METHOD PROTECTED FINAL allocate : BOOL
VAR_INPUT
	SizeOfStruct											: 	UDINT;	
END_VAR
IF SizeOfStruct = 0
THEN
	allocate												:= FALSE;
ELSIF pElement_Tmp = 0 
THEN
	pElement_Tmp											:= __NEW(BYTE, SizeOfStruct);
	MemSizeOfStruct											:= SizeOfStruct;
	IF TRUE
	THEN
		AdsLogHint('EngineeringToolbox | FB Quicksort | An instance allocated %s bytes from the dynamic memory of the ADS router memory pool', TO_STRING(MemSizeOfStruct));
	END_IF
	Allocate												:= TRUE;
ELSIF SizeOfStruct > MemSizeOfStruct
THEN
	__DELETE(pElement_Tmp);	
	pElement_Tmp											:= __NEW(BYTE, SizeOfStruct);
	MemSizeOfStruct											:= SizeOfStruct;
		IF TRUE
	THEN
		AdsLogWarn('EngineeringToolbox | FB Quicksort | SizeOfStruct increased and an instance has an additional %s bytes allocated from the dynamic memory of the ADS router memory pool', TO_STRING(MemSizeOfStruct));
	END_IF
	Allocate												:= TRUE;
ELSE
	Allocate												:= TRUE;	
END_IF
END_METHOD

METHOD byDINT : BOOL // returns true if sort ends successfully 
VAR_INPUT
	pData													: 	POINTER TO BYTE := 0;	// ADR(Array) 	
	SizeOfData												: 	UDINT := 0;				// SIZEOF(Array)
	pCompareElement											: 	POINTER TO BYTE := 0;	// ADR(Array[1].DINT)		
	SizeOfStruct											: 	UDINT := 0;				// SIZEOF(Array[1]) 	
END_VAR                                                 
VAR        
	pPivotElement											: 	POINTER TO DINT;		// Pivot value
	PivotElement											: 	DINT;					// Pivot value as DINT	
	pCmpElement												:	POINTER TO DINT;		// compare value
	                                					                            	
	endMainLoop												:	BOOL;					// End of main loop reached
	endSubLoop												:	BOOL;					// End of sub loop reached                                              
	ElementCount											:	DINT;					// No of array elements
	stackCount,left,right,i,j								:	DINT;					// running variables 	
	stack													:	ARRAY[1..32] OF UDINT;	// stack size 32 => ~1 Mio elements *)	
	                                					
	pElement_1												:	POINTER TO BYTE;		// Copy Pointer 1		
	pElement_2												:	POINTER TO BYTE;		// Copy Pointer 2

END_VAR
// ends with true in case of no error	                                    					 					
IF SizeOfStruct = 0 OR SizeOfData = 0
	OR pData = 0 OR pCompareElement = 0
THEN               					                                   					
	byDINT													:= FALSE;
	RETURN;   
ELSE
	byDINT													:= TRUE;                          					
END_IF                                  					
          
// calculate no. of Elements                                
ElementCount												:= TO_DINT(SizeOfData / SizeOfStruct);   		
			
// Quicksort                            					
// initial value of array size          					
left 														:= 1;				// first element
right 														:= ElementCount;	// last element 
stackCount 													:= 1;				// running variable 
                                        	
WHILE NOT endMainLoop DO							
	IF left < right THEN                	
		pPivotElement										:= pCompareElement + (SizeOfStruct * TO_UDINT(SHR(right+left,1)));
		PivotElement										:= pPivotElement^;
		i 													:= left -1;
		j 													:= right +1;
		endSubLoop 											:= FALSE;
		REPEAT
			IF SortInverse
			THEN	// sort descending	
				REPEAT	
					i 										:= i+1;	
					pCmpElement								:= pCompareElement + (SizeOfStruct * TO_UDINT(i-1));
				UNTIL (pCmpElement^ <= PivotElement) OR NOT (i < right)	END_REPEAT	
				REPEAT	
					j 										:= j-1;	
					pCmpElement								:= pCompareElement + (SizeOfStruct * TO_UDINT(j-1));
				UNTIL (pCmpElement^ >= PivotElement) OR NOT (j > left)	END_REPEAT		
			ELSE	// sort ascending
				REPEAT	
					i 										:= i+1;
					pCmpElement								:= pCompareElement + (SizeOfStruct * TO_UDINT(i-1));
				UNTIL (pCmpElement^ >= PivotElement)	OR NOT (i < right)	END_REPEAT;				
				REPEAT	
					j 										:= j-1;	
					pCmpElement								:= pCompareElement + (SizeOfStruct * TO_UDINT(j-1));
				UNTIL (pCmpElement^ <= PivotElement) OR NOT (j > left)	END_REPEAT;
			END_IF
			IF i >= j THEN
				endSubLoop									:= TRUE;
			ELSE                    					
				Allocate( SizeOfStruct);
				pElement_1									:= pData + (SizeOfStruct * TO_UDINT(j-1));
				pElement_2									:= pData + (SizeOfStruct * TO_UDINT(i-1));
				
				IF pElement_Tmp = 0 
					OR_ELSE MEMCPY(pElement_Tmp, pElement_1,	SizeOfStruct) = 0
					OR_ELSE MEMCPY(pElement_1,	pElement_2,		SizeOfStruct) = 0
					OR_ELSE MEMCPY(pElement_2,	pElement_Tmp,	SizeOfStruct) = 0
				THEN
					byDINT									:= FALSE;
					RETURN;	
				END_IF
	
			END_IF
		UNTIL endSubLoop END_REPEAT;		
		stack[stackCount] 									:= TO_UDINT(right); 	// save right in stack			
		IF stackCount < 32              					
		THEN                            					
			stackCount 										:= stackCount +1;
		ELSE															// Error stack Limit    
			endMainLoop 									:= TRUE;
			byDINT											:= FALSE;			
		END_IF                          					
		right 												:= MAX(left, i-1);
	ELSE                                
		IF stackCount = 1 THEN          
			endMainLoop 									:= TRUE;
		ELSE                            					
			left 											:= right+1;       
			stackCount 										:= stackCount -1;	// load from stack
			right											:= TO_DINT(stack[stackCount]);
		END_IF
	END_IF
END_WHILE
END_METHOD

METHOD byDINT_Bubble : BOOL // returns true if sort ends successfully 
VAR_INPUT	
	pData													:	POINTER TO BYTE;// ADR(Array) 			
	SizeOfData												:	UDINT;			// SIZEOF(Array)
	pCompareElement											:	POINTER TO BYTE;// ADR(Array[1].DINT)		
	SizeOfStruct											:	UDINT;			// SIZEOF(Array[1]) 			
END_VAR                                 					                
VAR                                     					                
	Run  													:	DINT;			// main loop
  	Index													:	DINT;			// sub loop 	
	ElementCount											:	DINT;			
	                                    					
	CompareElement_1										:	DINT;					
	CompareElement_2										:	DINT;					
	pCompareElement_1										:	POINTER TO DINT;		
	pCompareElement_2										:	POINTER TO DINT;
		                                					                        
	pElement_1												:	POINTER TO BYTE;		
	pElement_2												:	POINTER TO BYTE;		
END_VAR
// ends with true in case of no error	                                    					 					
IF SizeOfStruct = 0 OR SizeOfData = 0
	OR pData = 0 OR pCompareElement = 0
THEN               					                                   					
	byDINT_Bubble											:= FALSE;
	RETURN;   
ELSE
	byDINT_Bubble											:= TRUE;                          					
END_IF    

// Bubblesort Routine
// Code saving 
	
// calculate no. of Elements                                
ElementCount												:= TO_DINT(SizeOfData / SizeOfStruct);  

// bubblesort 
FOR Run := 1 TO TO_DINT(ElementCount) - 1 DO
    FOR Index := ElementCount - 1 TO Run BY -1 DO
		// get element x for compare 
		pCompareElement_1				:=	pCompareElement + (SizeOfStruct * TO_UDINT(Index));
		CompareElement_1				:=	pCompareElement_1^;
		// get element x-1 for compare 
		pCompareElement_2				:=	pCompareElement + (SizeOfStruct * TO_UDINT(Index-1));
		CompareElement_2 				:=	pCompareElement_2^;
		// switch by useing temporary memory 
		IF ((	CompareElement_1 < CompareElement_2) AND NOT SortInverse)
			OR((CompareElement_1 > CompareElement_2) AND SortInverse)
		THEN
			// get pointer for MEMCPY 
			Allocate(SizeOfStruct);
			pElement_1					:= pData + SizeOfStruct * TO_UDINT(Index);
			pElement_2					:= pData + SizeOfStruct * TO_UDINT(Index-1);
			
	
			IF pElement_Tmp = 0 
				OR_ELSE MEMCPY(pElement_Tmp, pElement_1,	SizeOfStruct) = 0
				OR_ELSE MEMCPY(pElement_1,	pElement_2,		SizeOfStruct) = 0
				OR_ELSE MEMCPY(pElement_2,	pElement_Tmp,	SizeOfStruct) = 0
			THEN
				byDINT_Bubble		:= FALSE;
				EXIT;												
			END_IF

      END_IF
	END_FOR
END_FOR
END_METHOD

METHOD byINT : BOOL // returns true if sort ends successfully 
VAR_INPUT
	pData													: 	POINTER TO BYTE := 0;	// ADR(Array) 	
	SizeOfData												: 	UDINT := 0;				// SIZEOF(Array)
	pCompareElement											: 	POINTER TO BYTE := 0;	// ADR(Array[1].INT)		
	SizeOfStruct											: 	UDINT := 0;				// SIZEOF(Array[1]) 	
END_VAR                                                 
VAR        
	pPivotElement											: 	POINTER TO INT;			// Pivot value
	PivotElement											: 	INT;					// Pivot value as INT	
	pCmpElement												:	POINTER TO INT;			// compare value
	                                					                            	
	endMainLoop												:	BOOL;					// End of main loop reached
	endSubLoop												:	BOOL;					// End of sub loop reached                                              
	ElementCount											:	DINT;					// No of array elements
	stackCount,left,right,i,j								:	DINT;					// running variables 	
	stack													:	ARRAY[1..32] OF UDINT;	// stack size 32 => ~1 Mio elements *)	
	                                					
	pElement_1												:	POINTER TO BYTE;		// Copy Pointer 1		
	pElement_2												:	POINTER TO BYTE;		// Copy Pointer 2
END_VAR
// ends with true in case of no error	                                    					 					
IF SizeOfStruct = 0 OR SizeOfData = 0
	OR pData = 0 OR pCompareElement = 0
THEN               					                                   					
	byINT													:= FALSE;
	RETURN;   
ELSE
	byINT													:= TRUE;                          					
END_IF                                    					
        
// calculate no. of Elements                                
ElementCount												:= TO_DINT(SizeOfData / SizeOfStruct);   
                                					
// Quicksort                            					
// initial value of array size          					
left 														:= 1;				// first element
right 														:= ElementCount;	// last element 
stackCount 													:= 1;				// running variable 
                                        	
WHILE NOT endMainLoop DO							
	IF left < right THEN                	
		pPivotElement										:= pCompareElement + (SizeOfStruct * TO_UDINT(SHR(right+left,1)));
		PivotElement										:= pPivotElement^;
		i 													:= left -1;
		j 													:= right +1;
		endSubLoop 											:= FALSE;
		REPEAT
			IF SortInverse
			THEN	// sort descending	
				REPEAT	
					i 										:= i+1;	
					pCmpElement								:= pCompareElement + (SizeOfStruct * TO_UDINT(i-1));
				UNTIL (pCmpElement^ <= PivotElement) OR NOT (i < right)	END_REPEAT	
				REPEAT	
					j 										:= j-1;	
					pCmpElement								:= pCompareElement + (SizeOfStruct * TO_UDINT(j-1));
				UNTIL (pCmpElement^ >= PivotElement) OR NOT (j > left)	END_REPEAT		
			ELSE	// sort ascending
				REPEAT	
					i 										:= i+1;
					pCmpElement								:= pCompareElement + (SizeOfStruct * TO_UDINT(i-1));
				UNTIL (pCmpElement^ >= PivotElement)	OR NOT (i < right)	END_REPEAT;				
				REPEAT	
					j 										:= j-1;	
					pCmpElement								:= pCompareElement + (SizeOfStruct * TO_UDINT(j-1));
				UNTIL (pCmpElement^ <= PivotElement) OR NOT (j > left)	END_REPEAT;
			END_IF
			IF i >= j THEN
				endSubLoop									:= TRUE;
			ELSE                    					
				Allocate(SizeOfStruct);
				pElement_1									:= pData + (SizeOfStruct * TO_UDINT(j-1));
				pElement_2									:= pData + (SizeOfStruct * TO_UDINT(i-1));
				
				IF pElement_Tmp = 0 
					OR_ELSE MEMCPY(pElement_Tmp, pElement_1,	SizeOfStruct) = 0
					OR_ELSE MEMCPY(pElement_1,	pElement_2,		SizeOfStruct) = 0
					OR_ELSE MEMCPY(pElement_2,	pElement_Tmp,	SizeOfStruct) = 0
				THEN
					byINT									:= FALSE;
					RETURN;	
				END_IF
	
			END_IF
		UNTIL endSubLoop END_REPEAT;		
		stack[stackCount] 									:= TO_UDINT(right); 	// save right in stack			
		IF stackCount < 32              					
		THEN                            					
			stackCount 										:= stackCount +1;
		ELSE															// Error stack Limit    
			endMainLoop 									:= TRUE;
			byINT											:= FALSE;			
		END_IF                          					
		right 												:= MAX(left, i-1);
	ELSE                                
		IF stackCount = 1 THEN          
			endMainLoop 									:= TRUE;
		ELSE                            					
			left 											:= right+1;       
			stackCount 										:= stackCount -1;	// load from stack
			right											:= TO_DINT(stack[stackCount]);
		END_IF
	END_IF
END_WHILE
END_METHOD

METHOD byLREAL : BOOL // returns true if sort ends successfully 
VAR_INPUT
	pData													: 	POINTER TO BYTE := 0;	// ADR(Array) 	
	SizeOfData												: 	UDINT := 0;				// SIZEOF(Array)
	pCompareElement											: 	POINTER TO BYTE := 0;	// ADR(Array[1].LREAL)		
	SizeOfStruct											: 	UDINT := 0;				// SIZEOF(Array[1]) 	
END_VAR                                                 
VAR        
	pPivotElement											: 	POINTER TO LREAL;		// Pivot value	
	PivotElement											: 	LREAL;					// Pivot value as LREAL
	pCmpElement												:	POINTER TO LREAL;		// compare value
	                                					                            	
	endMainLoop												:	BOOL;					// End of main loop reached
	endSubLoop												:	BOOL;					// End of sub loop reached                                              
	ElementCount											:	DINT;					// No of array elements
	stackCount,left,right,i,j								:	DINT;					// running variables 	
	stack													:	ARRAY[1..32] OF UDINT;	// stack size 32 => ~1 Mio elements *)	
	                                					
	pElement_1												:	POINTER TO BYTE;		// Copy Pointer 1		
	pElement_2												:	POINTER TO BYTE;		// Copy Pointer 2
	
END_VAR
// ends with true in case of no error	                                    					 					
IF SizeOfStruct = 0 OR SizeOfData = 0
	OR pData = 0 OR pCompareElement = 0
THEN               					                                   					
	byLREAL													:= FALSE;
	RETURN;   
ELSE
	byLREAL													:= TRUE;                          					
END_IF                                 					
            
// calculate no. of Elements                                
ElementCount												:= TO_DINT(SizeOfData / SizeOfStruct);   
                            					
// Quicksort                            					
// initial value of array size          					
left 														:= 1;				// first element
right 														:= ElementCount;	// last element 
stackCount 													:= 1;				// running variable 
                                        	
WHILE NOT endMainLoop DO							
	IF left < right THEN                	
		pPivotElement										:= pCompareElement + (SizeOfStruct * TO_UDINT(SHR(right+left,1))); // divide by 2
		PivotElement										:= pPivotElement^;
		i 													:= left -1;
		j 													:= right +1;
		endSubLoop 											:= FALSE;
		REPEAT
			IF SortInverse
			THEN	// sort descending	
				REPEAT	
					i 										:= i+1;	
					pCmpElement								:= pCompareElement + (SizeOfStruct * TO_UDINT(i-1));
				UNTIL (pCmpElement^ <= PivotElement) OR NOT (i < right)	END_REPEAT	
				REPEAT	
					j 										:= j-1;	
					pCmpElement								:= pCompareElement + (SizeOfStruct * TO_UDINT(j-1));
				UNTIL (pCmpElement^ >= PivotElement) OR NOT (j > left)	END_REPEAT		
			ELSE	// sort ascending
				REPEAT	
					i 										:= i+1;
					pCmpElement								:= pCompareElement + (SizeOfStruct * TO_UDINT(i-1));
				UNTIL (pCmpElement^ >= PivotElement)	OR NOT (i < right)	END_REPEAT;				
				REPEAT	
					j 										:= j-1;	
					pCmpElement								:= pCompareElement + (SizeOfStruct * TO_UDINT(j-1));
				UNTIL (pCmpElement^ <= PivotElement) OR NOT (j > left)	END_REPEAT;
			END_IF
			IF i >= j THEN
				endSubLoop									:= TRUE;
			ELSE                    					
				Allocate(SizeOfStruct);
				pElement_1									:= pData + (SizeOfStruct * TO_UDINT(j-1));
				pElement_2									:= pData + (SizeOfStruct * TO_UDINT(i-1));
				
				IF pElement_Tmp = 0 
					OR_ELSE MEMCPY(pElement_Tmp, pElement_1,	SizeOfStruct) = 0
					OR_ELSE MEMCPY(pElement_1,	pElement_2,		SizeOfStruct) = 0
					OR_ELSE MEMCPY(pElement_2,	pElement_Tmp,	SizeOfStruct) = 0
				THEN
					byLREAL									:= FALSE;
					RETURN;	
				END_IF

			END_IF
		UNTIL endSubLoop END_REPEAT;		
		stack[stackCount] 									:= TO_UDINT(right); 	// save right in stack			
		IF stackCount < 32              					
		THEN                            					
			stackCount 										:= stackCount +1;
		ELSE															// Error stack Limit    
			endMainLoop 									:= TRUE;
			byLREAL											:= FALSE;			
		END_IF                          					
		right 												:= MAX(left, i-1);
	ELSE                                
		IF stackCount = 1 THEN          
			endMainLoop 									:= TRUE;
		ELSE                            					
			left 											:= right+1;       
			stackCount 										:= stackCount -1;	// load from stack
			right											:= TO_DINT(stack[stackCount]);
		END_IF
	END_IF
END_WHILE
END_METHOD

METHOD byLTIME : BOOL // returns true if sort ends successfully 
VAR_INPUT
	pData													: 	POINTER TO BYTE := 0;	// ADR(Array) 	
	SizeOfData												: 	UDINT := 0;				// SIZEOF(Array)
	pCompareElement											: 	POINTER TO BYTE := 0;	// ADR(Array[1].LTIME)		
	SizeOfStruct											: 	UDINT := 0;				// SIZEOF(Array[1]) 	
END_VAR                                                 
VAR        
	pPivotElement											: 	POINTER TO LTIME;		// Pivot value	
	PivotElement											: 	LTIME;					// Pivot value as LTIME	
	pCmpElement												:	POINTER TO LTIME;		// compare value
	                                					                            	
	endMainLoop												:	BOOL;					// End of main loop reached
	endSubLoop												:	BOOL;					// End of sub loop reached                                              
	ElementCount											:	DINT;					// No of array elements
	stackCount,left,right,i,j								:	DINT;					// running variables 	
	stack													:	ARRAY[1..32] OF UDINT;	// stack size 32 => ~1 Mio elements *)	
	                                					
	pElement_1												:	POINTER TO BYTE;		// Copy Pointer 1		
	pElement_2												:	POINTER TO BYTE;		// Copy Pointer 2
END_VAR
// ends with true in case of no error	                                    					 					
IF SizeOfStruct = 0 OR SizeOfData = 0
	OR pData = 0 OR pCompareElement = 0
THEN               					                                   					
	byLTIME													:= FALSE;
	RETURN;   
ELSE
	byLTIME													:= TRUE;                          					
END_IF                                    					
             
// calculate no. of Elements                                
ElementCount												:= TO_DINT(SizeOfData / SizeOfStruct);   
                           					
// Quicksort                            					
// initial value of array size          					
left 														:= 1;				// first element
right 														:= ElementCount;	// last element 
stackCount 													:= 1;				// running variable 
                                        	
WHILE NOT endMainLoop DO							
	IF left < right THEN                	
		pPivotElement										:= pCompareElement + (SizeOfStruct * TO_UDINT(SHR(right+left,1)));
		PivotElement										:= pPivotElement^;
		i 													:= left -1;
		j 													:= right +1;
		endSubLoop 											:= FALSE;
		REPEAT
			IF SortInverse
			THEN	// sort descending	
				REPEAT	
					i 										:= i+1;	
					pCmpElement								:= pCompareElement + (SizeOfStruct * TO_UDINT(i-1));
				UNTIL (pCmpElement^ <= PivotElement) OR NOT (i < right)	END_REPEAT	
				REPEAT	
					j 										:= j-1;	
					pCmpElement								:= pCompareElement + (SizeOfStruct * TO_UDINT(j-1));
				UNTIL (pCmpElement^ >= PivotElement) OR NOT (j > left)	END_REPEAT		
			ELSE	// sort ascending
				REPEAT	
					i 										:= i+1;
					pCmpElement								:= pCompareElement + (SizeOfStruct * TO_UDINT(i-1));
				UNTIL (pCmpElement^ >= PivotElement)	OR NOT (i < right)	END_REPEAT;				
				REPEAT	
					j 										:= j-1;	
					pCmpElement								:= pCompareElement + (SizeOfStruct * TO_UDINT(j-1));
				UNTIL (pCmpElement^ <= PivotElement) OR NOT (j > left)	END_REPEAT;
			END_IF
			IF i >= j THEN
				endSubLoop									:= TRUE;
			ELSE                    					
				Allocate(SizeOfStruct);
				pElement_1									:= pData + (SizeOfStruct * TO_UDINT(j-1));
				pElement_2									:= pData + (SizeOfStruct * TO_UDINT(i-1));
				
				IF pElement_Tmp = 0 
					OR_ELSE MEMCPY(pElement_Tmp, pElement_1,	SizeOfStruct) = 0
					OR_ELSE MEMCPY(pElement_1,	pElement_2,		SizeOfStruct) = 0
					OR_ELSE MEMCPY(pElement_2,	pElement_Tmp,	SizeOfStruct) = 0
				THEN
					byLTIME									:= FALSE;
					RETURN;	
				END_IF

			END_IF
		UNTIL endSubLoop END_REPEAT;		
		stack[stackCount] 									:= TO_UDINT(right); 	// save right in stack			
		IF stackCount < 32              					
		THEN                            					
			stackCount 										:= stackCount +1;
		ELSE															// Error stack Limit    
			endMainLoop 									:= TRUE;
			byLTIME											:= FALSE;			
		END_IF                          					
		right 												:= MAX(left, i-1);
	ELSE                                
		IF stackCount = 1 THEN          
			endMainLoop 									:= TRUE;
		ELSE                            					
			left 											:= right+1;       
			stackCount 										:= stackCount -1;	// load from stack
			right											:= TO_DINT(stack[stackCount]);
		END_IF
	END_IF
END_WHILE
END_METHOD

METHOD byREAL : BOOL // returns true if sort ends successfully 
VAR_INPUT
	pData													: 	POINTER TO BYTE := 0;	// ADR(Array) 	
	SizeOfData												: 	UDINT := 0;				// SIZEOF(Array)
	pCompareElement											: 	POINTER TO BYTE := 0;	// ADR(Array[1].REAL)		
	SizeOfStruct											: 	UDINT := 0;				// SIZEOF(Array[1]) 	
END_VAR                                                 
VAR        
	pPivotElement											: 	POINTER TO REAL;		// Pivot value	
	PivotElement											: 	REAL;					// Pivot value as REAL	
	pCmpElement												:	POINTER TO REAL;		// compare value
	                                					                            	
	endMainLoop												:	BOOL;					// End of main loop reached
	endSubLoop												:	BOOL;					// End of sub loop reached                                              
	ElementCount											:	DINT;					// No of array elements
	stackCount,left,right,i,j								:	DINT;					// running variables 	
	stack													:	ARRAY[1..32] OF UDINT;	// stack size 32 => ~1 Mio elements *)	
	                                					
	pElement_1												:	POINTER TO BYTE;		// Copy Pointer 1		
	pElement_2												:	POINTER TO BYTE;		// Copy Pointer 2
END_VAR
// ends with true in case of no error	                                    					 					
IF SizeOfStruct = 0 OR SizeOfData = 0
	OR pData = 0 OR pCompareElement = 0
THEN               					                                   					
	byREAL													:= FALSE;
	RETURN;   
ELSE
	byREAL													:= TRUE;                          					
END_IF                                   					
          
// calculate no. of Elements                                
ElementCount												:= TO_DINT(SizeOfData / SizeOfStruct);   
                              					
// Quicksort                            					
// initial value of array size          					
left 														:= 1;				// first element
right 														:= ElementCount;	// last element 
stackCount 													:= 1;				// running variable 
                                        	
WHILE NOT endMainLoop DO							
	IF left < right THEN                	
		pPivotElement										:= pCompareElement + (SizeOfStruct * TO_UDINT(SHR(right+left,1)));
		PivotElement										:= pPivotElement^;
		i 													:= left -1;
		j 													:= right +1;
		endSubLoop 											:= FALSE;
		REPEAT
			IF SortInverse
			THEN	// sort descending	
				REPEAT	
					i 										:= i+1;	
					pCmpElement								:= pCompareElement + (SizeOfStruct * TO_UDINT(i-1));
				UNTIL (pCmpElement^ <= PivotElement) OR NOT (i < right)	END_REPEAT	
				REPEAT	
					j 										:= j-1;	
					pCmpElement								:= pCompareElement + (SizeOfStruct * TO_UDINT(j-1));
				UNTIL (pCmpElement^ >= PivotElement) OR NOT (j > left)	END_REPEAT		
			ELSE	// sort ascending
				REPEAT	
					i 										:= i+1;
					pCmpElement								:= pCompareElement + (SizeOfStruct * TO_UDINT(i-1));
				UNTIL (pCmpElement^ >= PivotElement)	OR NOT (i < right)	END_REPEAT;				
				REPEAT	
					j 										:= j-1;	
					pCmpElement								:= pCompareElement + (SizeOfStruct * TO_UDINT(j-1));
				UNTIL (pCmpElement^ <= PivotElement) OR NOT (j > left)	END_REPEAT;
			END_IF
			IF i >= j THEN
				endSubLoop									:= TRUE;
			ELSE                    					
				Allocate(SizeOfStruct);
				pElement_1									:= pData + (SizeOfStruct * TO_UDINT(j-1));
				pElement_2									:= pData + (SizeOfStruct * TO_UDINT(i-1));
				
				IF pElement_Tmp = 0 
					OR_ELSE MEMCPY(pElement_Tmp, pElement_1,	SizeOfStruct) = 0
					OR_ELSE MEMCPY(pElement_1,	pElement_2,		SizeOfStruct) = 0
					OR_ELSE MEMCPY(pElement_2,	pElement_Tmp,	SizeOfStruct) = 0
				THEN
					byREAL									:= FALSE;
					RETURN;	
				END_IF

			END_IF
		UNTIL endSubLoop END_REPEAT;		
		stack[stackCount] 									:= TO_UDINT(right); 	// save right in stack			
		IF stackCount < 32              					
		THEN                            					
			stackCount 										:= stackCount +1;
		ELSE															// Error stack Limit    
			endMainLoop 									:= TRUE;
			byREAL											:= FALSE;			
		END_IF                          					
		right 												:= MAX(left, i-1);
	ELSE                                
		IF stackCount = 1 THEN          
			endMainLoop 									:= TRUE;
		ELSE                            					
			left 											:= right+1;       
			stackCount 										:= stackCount -1;	// load from stack
			right											:= TO_DINT(stack[stackCount]);
		END_IF
	END_IF
END_WHILE
END_METHOD

METHOD bySTRING : BOOL // returns true if sort ends successfully 
VAR_INPUT
	pData													: 	POINTER TO BYTE := 0;	// ADR(Array) 	
	SizeOfData												: 	UDINT := 0;				// SIZEOF(Array)
	pCompareElement											: 	POINTER TO BYTE := 0;	// ADR(Array[1].STRING)		
	SizeOfStruct											: 	UDINT := 0;				// SIZEOF(Array[1]) 	
END_VAR                                                                                        
VAR        
	pPivotElement											: 	POINTER TO STRING(MAX_STRING_LENGTH);	// Pivot value
	pCmpElement												:	POINTER TO STRING(MAX_STRING_LENGTH);	// compare value
	PivotElement											:	BYTE; 					// Pivot value	
	CompareElement											:	BYTE; 					// compare value
                               					                            	
	endMainLoop												:	BOOL;					// End of main loop reached
	endSubLoop												:	BOOL;					// End of sub loop reached                                              
	ElementCount											:	DINT;					// No of array elements
	stackCount,left,right,i,j,k								:	DINT;					// running variables 	
	stack													:	ARRAY[1..32] OF UDINT;	// stack size 32 => ~1 Mio elements *)	
	                                					
	pElement_1												:	POINTER TO BYTE;		// Copy Pointer 1		
	pElement_2												:	POINTER TO BYTE;		// Copy Pointer 2
END_VAR
// ends with true in case of no error	                                    					 					
IF SizeOfStruct = 0 OR SizeOfData = 0
	OR pData = 0 OR pCompareElement = 0
THEN               					                                   					
	bySTRING												:= FALSE;
	RETURN;   
ELSE
	bySTRING												:= TRUE;                          					
END_IF                                 					
          
// calculate no. of Elements                                
ElementCount												:= TO_DINT(SizeOfData / SizeOfStruct);   
                              					
// Quicksort                            					
// initial value of array size          					
left 														:= 1;				// first element
right 														:= ElementCount;	// last element 
stackCount 													:= 1;				// running variable 
                                        	
WHILE NOT endMainLoop DO							
	IF left < right THEN                	
		pPivotElement										:= pCompareElement + (SizeOfStruct * TO_UDINT(SHR(right+left,1)));
		i 													:= left -1;
		j 													:= right +1;
		endSubLoop 											:= FALSE;
		REPEAT
			IF SortInverse
			THEN	// sort descending	
				REPEAT	
					i 										:= i+1;	
					pCmpElement								:= pCompareElement + (SizeOfStruct * TO_UDINT(i-1));
					FOR k := 1 TO MAX_STRING_LENGTH DO // Find unequal char
						// element 1,2 to upper char 	https://www.uni-due.de/hummell/infos/ascii/
						IF pCmpElement^[k] = 0 
							AND IgnoreBlank
						THEN
							CompareElement					:= 127;
						ELSE
							CompareElement					:= SEL(pCmpElement^[k] >= 97(*a*)	AND_THEN pCmpElement^[k] <= 122(*z*), 	pCmpElement^[k],pCmpElement^[k] - 32);		// a --> A
						END_IF						
						IF pPivotElement^[k] = 0 
							AND IgnoreBlank
						THEN
							PivotElement					:= 127;
						ELSE
							PivotElement					:= SEL(pPivotElement^[k] >= 97(*a*) AND_THEN pPivotElement^[k] <= 122(*z*), pPivotElement^[k], 	pPivotElement^[k] - 32);// a --> A
						END_IF
						// Find unequal char
						IF CompareElement <> PivotElement
							OR CompareElement = 0
							OR PivotElement = 0
						THEN
							EXIT;
						END_IF
					END_FOR
				UNTIL (CompareElement <= PivotElement) OR NOT (i < right)	END_REPEAT	
				REPEAT	
					j 										:= j-1;	
					pCmpElement								:= pCompareElement + (SizeOfStruct * TO_UDINT(j-1));
					FOR k := 0 TO MAX_STRING_LENGTH DO // Find unequal char
						// element 1,2 to upper char 	https://www.uni-due.de/hummell/infos/ascii/
						IF pCmpElement^[k] = 0 
							AND IgnoreBlank
						THEN
							CompareElement					:= 127;
						ELSE
							CompareElement					:= SEL(pCmpElement^[k] >= 97(*a*)	AND_THEN pCmpElement^[k] <= 122(*z*), 	pCmpElement^[k],pCmpElement^[k] - 32);		// a --> A
						END_IF
						IF pPivotElement^[k] = 0 
							AND IgnoreBlank
						THEN
							PivotElement					:= 127;
						ELSE
							PivotElement					:= SEL(pPivotElement^[k] >= 97(*a*) AND_THEN pPivotElement^[k] <= 122(*z*), pPivotElement^[k], 	pPivotElement^[k] - 32);// a --> A
						END_IF
						// Find unequal char
						IF CompareElement <> PivotElement
							OR CompareElement = 0
							OR PivotElement = 0
						THEN
							EXIT;
						END_IF
					END_FOR
				UNTIL (CompareElement >= PivotElement) OR NOT (j > left)	END_REPEAT		
			ELSE	// sort ascending
				REPEAT	
					i 										:= i+1;
					pCmpElement								:= pCompareElement + (SizeOfStruct * TO_UDINT(i-1));
					FOR k := 0 TO MAX_STRING_LENGTH DO // Find unequal char
						// element 1,2 to upper char 	https://www.uni-due.de/hummell/infos/ascii/
						IF pCmpElement^[k] = 0 
							AND IgnoreBlank
						THEN
							CompareElement					:= 127;
						ELSE
							CompareElement					:= SEL(pCmpElement^[k] >= 97(*a*)	AND_THEN pCmpElement^[k] <= 122(*z*), 	pCmpElement^[k],pCmpElement^[k] - 32);		// a --> A
						END_IF
						IF pPivotElement^[k] = 0 
							AND IgnoreBlank
						THEN
							PivotElement					:= 127;
						ELSE
							PivotElement					:= SEL(pPivotElement^[k] >= 97(*a*) AND_THEN pPivotElement^[k] <= 122(*z*), pPivotElement^[k], 	pPivotElement^[k] - 32);// a --> A
						END_IF
						// Find unequal char
						IF CompareElement <> PivotElement
							OR CompareElement = 0
							OR PivotElement = 0
						THEN
							EXIT;
						END_IF
					END_FOR
				UNTIL (CompareElement >= PivotElement)	OR NOT (i < right)	END_REPEAT;				
				REPEAT	
					j 										:= j-1;	
					pCmpElement								:= pCompareElement + (SizeOfStruct * TO_UDINT(j-1));
					FOR k := 0 TO MAX_STRING_LENGTH DO // Find unequal char
						// element 1,2 to upper char 	https://www.uni-due.de/hummell/infos/ascii/
						IF pCmpElement^[k] = 0 
							AND IgnoreBlank
						THEN	
							CompareElement					:= 127;
						ELSE
							CompareElement					:= SEL(pCmpElement^[k] >= 97(*a*)	AND_THEN pCmpElement^[k] <= 122(*z*), 	pCmpElement^[k],pCmpElement^[k] - 32);		// a --> A
						END_IF
						IF pPivotElement^[k] = 0
							AND IgnoreBlank 
						THEN
							PivotElement					:= 127;
						ELSE
							PivotElement					:= SEL(pPivotElement^[k] >= 97(*a*) AND_THEN pPivotElement^[k] <= 122(*z*), pPivotElement^[k], 	pPivotElement^[k] - 32);// a --> A
						END_IF
						// Find unequal char
						IF CompareElement <> PivotElement
							OR CompareElement = 0
							OR PivotElement = 0
						THEN
							EXIT;
						END_IF
					END_FOR
				UNTIL (CompareElement <= PivotElement) OR NOT (j > left)	END_REPEAT;
			END_IF
			IF i >= j THEN
				endSubLoop									:= TRUE;
			ELSE                    					
				Allocate(SizeOfStruct);
				pElement_1									:= pData + (SizeOfStruct * TO_UDINT(j-1));
				pElement_2									:= pData + (SizeOfStruct * TO_UDINT(i-1));
				
				IF pElement_Tmp = 0 
					OR_ELSE MEMCPY(pElement_Tmp, pElement_1,	SizeOfStruct) = 0
					OR_ELSE MEMCPY(pElement_1,	pElement_2,		SizeOfStruct) = 0
					OR_ELSE MEMCPY(pElement_2,	pElement_Tmp,	SizeOfStruct) = 0
				THEN
					bySTRING								:= FALSE;
					RETURN;	
				END_IF

			END_IF
		UNTIL endSubLoop END_REPEAT;		
		stack[stackCount] 									:= TO_UDINT(right); 	// save right in stack			
		IF stackCount < 32              					
		THEN                            					
			stackCount 										:= stackCount +1;
		ELSE															// Error stack Limit    
			endMainLoop 									:= TRUE;
			bySTRING										:= FALSE;			
		END_IF                          					
		right 												:= MAX(left, i-1);
	ELSE                                
		IF stackCount = 1 THEN          
			endMainLoop 									:= TRUE;
		ELSE                            					
			left 											:= right+1;       
			stackCount 										:= stackCount -1;	// load from stack
			right											:= TO_DINT(stack[stackCount]);
		END_IF
	END_IF
END_WHILE
END_METHOD

METHOD byTIME : BOOL // returns true if sort ends successfully 
VAR_INPUT
	pData													: 	POINTER TO BYTE := 0;	// ADR(Array) 	
	SizeOfData												: 	UDINT := 0;				// SIZEOF(Array)
	pCompareElement											: 	POINTER TO BYTE := 0;	// ADR(Array[1].TIME)		
	SizeOfStruct											: 	UDINT := 0;				// SIZEOF(Array[1]) 	
END_VAR                                                 
VAR        
	pPivotElement											: 	POINTER TO TIME;		// Pivot value
	PivotElement											: 	TIME;					// Pivot value as TIME	
	pCmpElement												:	POINTER TO TIME;		// compare value
	                                					                            	
	endMainLoop												:	BOOL;					// End of main loop reached
	endSubLoop												:	BOOL;					// End of sub loop reached                                              
	ElementCount											:	DINT;					// No of array elements
	stackCount,left,right,i,j								:	DINT;					// running variables 	
	stack													:	ARRAY[1..32] OF UDINT;	// stack size 32 => ~1 Mio elements *)	
	                                					
	pElement_1												:	POINTER TO BYTE;		// Copy Pointer 1		
	pElement_2												:	POINTER TO BYTE;		// Copy Pointer 2
END_VAR
// ends with true in case of no error	                                    					 					
IF SizeOfStruct = 0 OR SizeOfData = 0
	OR pData = 0 OR pCompareElement = 0
THEN               					                                   					
	byTIME													:= FALSE;
	RETURN;   
ELSE
	byTIME													:= TRUE;                          					
END_IF   

// calculate no. of Elements                                
ElementCount												:= TO_DINT(SizeOfData / SizeOfStruct);                                   					
                                        					
// Quicksort                            					
// initial value of array size          					
left 														:= 1;				// first element
right 														:= ElementCount;	// last element 
stackCount 													:= 1;				// running variable 
                                        	
WHILE NOT endMainLoop DO							
	IF left < right THEN                	
		pPivotElement										:= pCompareElement + (SizeOfStruct * TO_UDINT(SHR(right+left,1)));
		PivotElement										:= pPivotElement^;
		i 													:= left -1;
		j 													:= right +1;
		endSubLoop 											:= FALSE;
		REPEAT
			IF SortInverse
			THEN	// sort descending	
				REPEAT	
					i 										:= i+1;	
					pCmpElement								:= pCompareElement + (SizeOfStruct * TO_UDINT(i-1));
				UNTIL (pCmpElement^ <= PivotElement) OR NOT (i < right)	END_REPEAT	
				REPEAT	
					j 										:= j-1;	
					pCmpElement								:= pCompareElement + (SizeOfStruct * TO_UDINT(j-1));
				UNTIL (pCmpElement^ >= PivotElement) OR NOT (j > left)	END_REPEAT		
			ELSE	// sort ascending
				REPEAT	
					i 										:= i+1;
					pCmpElement								:= pCompareElement + (SizeOfStruct * TO_UDINT(i-1));
				UNTIL (pCmpElement^ >= PivotElement)	OR NOT (i < right)	END_REPEAT;				
				REPEAT	
					j 										:= j-1;	
					pCmpElement								:= pCompareElement + (SizeOfStruct * TO_UDINT(j-1));
				UNTIL (pCmpElement^ <= PivotElement) OR NOT (j > left)	END_REPEAT;
			END_IF
			IF i >= j THEN
				endSubLoop									:= TRUE;
			ELSE                    					
				Allocate(SizeOfStruct);
				pElement_1									:= pData + (SizeOfStruct * TO_UDINT(j-1));
				pElement_2									:= pData + (SizeOfStruct * TO_UDINT(i-1));
				
				IF pElement_Tmp = 0 
					OR_ELSE MEMCPY(pElement_Tmp, pElement_1,	SizeOfStruct) = 0
					OR_ELSE MEMCPY(pElement_1,	pElement_2,		SizeOfStruct) = 0
					OR_ELSE MEMCPY(pElement_2,	pElement_Tmp,	SizeOfStruct) = 0
				THEN
					byTIME									:= FALSE;
					RETURN;	
				END_IF

			END_IF
		UNTIL endSubLoop END_REPEAT;		
		stack[stackCount] 									:= TO_UDINT(right); 	// save right in stack			
		IF stackCount < 32              					
		THEN                            					
			stackCount 										:= stackCount +1;
		ELSE															// Error stack Limit    
			endMainLoop 									:= TRUE;
			byTIME											:= FALSE;			
		END_IF                          					
		right 												:= MAX(left, i-1);
	ELSE                                
		IF stackCount = 1 THEN          
			endMainLoop 									:= TRUE;
		ELSE                            					
			left 											:= right+1;       
			stackCount 										:= stackCount -1;	// load from stack
			right											:= TO_DINT(stack[stackCount]);
		END_IF
	END_IF
END_WHILE
END_METHOD

METHOD byUINT : BOOL // returns true if sort ends successfully 
VAR_INPUT
	pData													: 	POINTER TO BYTE := 0;	// ADR(Array) 	
	SizeOfData												: 	UDINT := 0;				// SIZEOF(Array)
	pCompareElement											: 	POINTER TO BYTE := 0;	// ADR(Array[1].UINT)		
	SizeOfStruct											: 	UDINT := 0;				// SIZEOF(Array[1]) 	
END_VAR                                                 
VAR        
	pPivotElement											: 	POINTER TO UINT;		// Pivot value	
	PivotElement											: 	UINT;					// Pivot value as UINT	
	pCmpElement												:	POINTER TO UINT;		// compare value
	                                					                            	
	endMainLoop												:	BOOL;					// End of main loop reached
	endSubLoop												:	BOOL;					// End of sub loop reached                                              
	ElementCount											:	DINT;					// No of array elements
	stackCount,left,right,i,j								:	DINT;					// running variables 	
	stack													:	ARRAY[1..32] OF UDINT;	// stack size 32 => ~1 Mio elements *)	
	                                					
	pElement_1												:	POINTER TO BYTE;		// Copy Pointer 1		
	pElement_2												:	POINTER TO BYTE;		// Copy Pointer 2
END_VAR
// ends with true in case of no error	                                    					 					
IF SizeOfStruct = 0 OR SizeOfData = 0
	OR pData = 0 OR pCompareElement = 0
THEN               					                                   					
	byUINT													:= FALSE;
	RETURN;   
ELSE
	byUINT													:= TRUE;                          					
END_IF     

// calculate no. of Elements                                
ElementCount												:= TO_DINT(SizeOfData / SizeOfStruct);                                 					
                                        					
// Quicksort                            					
// initial value of array size          					
left 														:= 1;				// first element
right 														:= ElementCount;	// last element 
stackCount 													:= 1;				// running variable 
                                        	
WHILE NOT endMainLoop DO							
	IF left < right THEN                	
		pPivotElement										:= pCompareElement + (SizeOfStruct * TO_UDINT(SHR(right+left,1)));
		PivotElement										:= pPivotElement^;
		i 													:= left -1;
		j 													:= right +1;
		endSubLoop 											:= FALSE;
		REPEAT
			IF SortInverse
			THEN	// sort descending	
				REPEAT	
					i 										:= i+1;	
					pCmpElement								:= pCompareElement + (SizeOfStruct * TO_UDINT(i-1));
				UNTIL (pCmpElement^ <= PivotElement) OR NOT (i < right)	END_REPEAT	
				REPEAT	
					j 										:= j-1;	
					pCmpElement								:= pCompareElement + (SizeOfStruct * TO_UDINT(j-1));
				UNTIL (pCmpElement^ >= PivotElement) OR NOT (j > left)	END_REPEAT		
			ELSE	// sort ascending
				REPEAT	
					i 										:= i+1;
					pCmpElement								:= pCompareElement + (SizeOfStruct * TO_UDINT(i-1));
				UNTIL (pCmpElement^ >= PivotElement)	OR NOT (i < right)	END_REPEAT;				
				REPEAT	
					j 										:= j-1;	
					pCmpElement								:= pCompareElement + (SizeOfStruct * TO_UDINT(j-1));
				UNTIL (pCmpElement^ <= PivotElement) OR NOT (j > left)	END_REPEAT;
			END_IF
			IF i >= j THEN
				endSubLoop									:= TRUE;
			ELSE                    					
				Allocate(SizeOfStruct);
				pElement_1									:= pData + (SizeOfStruct * TO_UDINT(j-1));
				pElement_2									:= pData + (SizeOfStruct * TO_UDINT(i-1));
				
				IF pElement_Tmp = 0 
					OR_ELSE MEMCPY(pElement_Tmp, pElement_1,	SizeOfStruct) = 0
					OR_ELSE MEMCPY(pElement_1,	pElement_2,		SizeOfStruct) = 0
					OR_ELSE MEMCPY(pElement_2,	pElement_Tmp,	SizeOfStruct) = 0
				THEN
					byUINT									:= FALSE;
					RETURN;	
				END_IF

			END_IF
		UNTIL endSubLoop END_REPEAT;		
		stack[stackCount] 									:= TO_UDINT(right); 	// save right in stack			
		IF stackCount < 32              					
		THEN                            					
			stackCount 										:= stackCount +1;
		ELSE															// Error stack Limit    
			endMainLoop 									:= TRUE;
			byUINT											:= FALSE;			
		END_IF                          					
		right 												:= MAX(left, i-1);
	ELSE                                
		IF stackCount = 1 THEN          
			endMainLoop 									:= TRUE;
		ELSE                            					
			left 											:= right+1;       
			stackCount 										:= stackCount -1;	// load from stack
			right											:= TO_DINT(stack[stackCount]);
		END_IF
	END_IF
END_WHILE
END_METHOD

METHOD byUSINT : BOOL // returns true if sort ends successfully 
VAR_INPUT
	pData													: 	POINTER TO BYTE := 0;	// ADR(Array) 	
	SizeOfData												: 	UDINT := 0;				// SIZEOF(Array)
	pCompareElement											: 	POINTER TO BYTE := 0;	// ADR(Array[1].USINT)		
	SizeOfStruct											: 	UDINT := 0;				// SIZEOF(Array[1]) 	
END_VAR                                                 
VAR        
	pPivotElement											: 	POINTER TO USINT;		// Pivot value	
	PivotElement											: 	USINT;					// Pivot value as USINT
	pCmpElement												:	POINTER TO USINT;		// compare value
	                                					                            	
	endMainLoop												:	BOOL;					// End of main loop reached
	endSubLoop												:	BOOL;					// End of sub loop reached                                              
	ElementCount											:	DINT;					// No of array elements
	stackCount,left,right,i,j								:	DINT;					// running variables 	
	stack													:	ARRAY[1..32] OF UDINT;	// stack size 32 => ~1 Mio elements *)	
	                                					
	pElement_1												:	POINTER TO BYTE;		// Copy Pointer 1		
	pElement_2												:	POINTER TO BYTE;		// Copy Pointer 2
END_VAR
// ends with true in case of no error	                                    					 					
IF SizeOfStruct = 0 OR SizeOfData = 0
	OR pData = 0 OR pCompareElement = 0
THEN               					                                   					
	byUSINT													:= FALSE;
	RETURN;   
ELSE
	byUSINT													:= TRUE;                          					
END_IF    

// calculate no. of Elements                                
ElementCount												:= TO_DINT(SizeOfData / SizeOfStruct);                               					
                                        					
// Quicksort                            					
// initial value of array size          					
left 														:= 1;				// first element
right 														:= ElementCount;	// last element 
stackCount 													:= 1;				// running variable 
                                        	
WHILE NOT endMainLoop DO							
	IF left < right THEN                	
		pPivotElement										:= pCompareElement + (SizeOfStruct * TO_UDINT(SHR(right+left,1)));
		PivotElement										:= pPivotElement^;
		i 													:= left -1;
		j 													:= right +1;
		endSubLoop 											:= FALSE;
		REPEAT
			IF SortInverse
			THEN	// sort descending	
				REPEAT	
					i 										:= i+1;	
					pCmpElement								:= pCompareElement + (SizeOfStruct * TO_UDINT(i-1));
				UNTIL (pCmpElement^ <= PivotElement) OR NOT (i < right)	END_REPEAT	
				REPEAT	
					j 										:= j-1;	
					pCmpElement								:= pCompareElement + (SizeOfStruct * TO_UDINT(j-1));
				UNTIL (pCmpElement^ >= PivotElement) OR NOT (j > left)	END_REPEAT		
			ELSE	// sort ascending
				REPEAT	
					i 										:= i+1;
					pCmpElement								:= pCompareElement + (SizeOfStruct * TO_UDINT(i-1));
				UNTIL (pCmpElement^ >= PivotElement)	OR NOT (i < right)	END_REPEAT;				
				REPEAT	
					j 										:= j-1;	
					pCmpElement								:= pCompareElement + (SizeOfStruct * TO_UDINT(j-1));
				UNTIL (pCmpElement^ <= PivotElement) OR NOT (j > left)	END_REPEAT;
			END_IF
			IF i >= j THEN
				endSubLoop									:= TRUE;
			ELSE                    					
				Allocate(SizeOfStruct);
				pElement_1									:= pData + (SizeOfStruct * TO_UDINT(j-1));
				pElement_2									:= pData + (SizeOfStruct * TO_UDINT(i-1));
				
				IF pElement_Tmp = 0 
					OR_ELSE MEMCPY(pElement_Tmp, pElement_1,	SizeOfStruct) = 0
					OR_ELSE MEMCPY(pElement_1,	pElement_2,		SizeOfStruct) = 0
					OR_ELSE MEMCPY(pElement_2,	pElement_Tmp,	SizeOfStruct) = 0
				THEN
					byUSINT									:= FALSE;
					RETURN;	
				END_IF

			END_IF
		UNTIL endSubLoop END_REPEAT;		
		stack[stackCount] 									:= TO_UDINT(right); 	// save right in stack			
		IF stackCount < 32              					
		THEN                            					
			stackCount 										:= stackCount +1;
		ELSE															// Error stack Limit    
			endMainLoop 									:= TRUE;
			byUSINT											:= FALSE;			
		END_IF                          					
		right 												:= MAX(left, i-1);
	ELSE                                
		IF stackCount = 1 THEN          
			endMainLoop 									:= TRUE;
		ELSE                            					
			left 											:= right+1;       
			stackCount 										:= stackCount -1;	// load from stack
			right											:= TO_DINT(stack[stackCount]);
		END_IF
	END_IF
END_WHILE
END_METHOD

METHOD byWSTRING : BOOL // returns true if sort ends successfully 
VAR_INPUT
	pData													: 	POINTER TO BYTE := 0;	// ADR(Array) 	
	SizeOfData												: 	UDINT := 0;				// SIZEOF(Array)
	pCompareElement											: 	POINTER TO BYTE := 0;	// ADR(Array[1].WSTRING)		
	SizeOfStruct											: 	UDINT := 0;				// SIZEOF(Array[1]) 	
END_VAR                                                                                            
VAR        
	pPivotElement											: 	POINTER TO WSTRING(MAX_WSTRING_LENGTH);	// Pivot value	
	pCmpElement												:	POINTER TO WSTRING(MAX_WSTRING_LENGTH);	// compare value
	PivotElement											:	WORD; 					// Pivot value	
	CompareElement											:	WORD; 					// compare value
	                                					                            	
	endMainLoop												:	BOOL;					// End of main loop reached
	endSubLoop												:	BOOL;					// End of sub loop reached                                              
	ElementCount											:	DINT;					// No of array elements
	stackCount,left,right,i,j,k								:	DINT;					// running variables 	
	stack													:	ARRAY[1..32] OF UDINT;	// stack size 32 => ~1 Mio elements *)	
	                                					
	pElement_1												:	POINTER TO BYTE;		// Copy Pointer 1		
	pElement_2												:	POINTER TO BYTE;		// Copy Pointer 2
END_VAR
// ends with true in case of no error	                                    					 					
IF SizeOfStruct = 0 OR SizeOfData = 0
	OR pData = 0 OR pCompareElement = 0
THEN               					                                   					
	byWSTRING												:= FALSE;
	RETURN;   
ELSE
	byWSTRING												:= TRUE;                          					
END_IF                                   					
            
// calculate no. of Elements                                
ElementCount												:= TO_DINT(SizeOfData / SizeOfStruct);   
                            					
// Quicksort                            					
// initial value of array size          					
left 														:= 1;				// first element
right 														:= ElementCount;	// last element 
stackCount 													:= 1;				// running variable 
                                        	
WHILE NOT endMainLoop DO							
	IF left < right THEN                	
		pPivotElement										:= pCompareElement + (SizeOfStruct * TO_UDINT(SHR(right+left,1)));
		i 													:= left -1;
		j 													:= right +1;
		endSubLoop 											:= FALSE;
		REPEAT
			IF SortInverse
			THEN	// sort descending	
				REPEAT	
					i 										:= i+1;	
					pCmpElement								:= pCompareElement + (SizeOfStruct * TO_UDINT(i-1));
					FOR k := 0 TO MAX_WSTRING_LENGTH DO // Find unequal char
						// element 1,2 to upper char 	https://www.uni-due.de/hummell/infos/ascii/
						IF pCmpElement^[k] = 0 
							AND IgnoreBlank
						THEN
							CompareElement					:= 127;
						ELSE
							CompareElement					:= SEL(pCmpElement^[k] >= 97(*a*)	AND_THEN pCmpElement^[k] <= 122(*z*), 	pCmpElement^[k],pCmpElement^[k] - 32);		// a --> A
						END_IF
						IF pPivotElement^[k] = 0 
							AND IgnoreBlank
						THEN
							PivotElement					:= 127;
						ELSE
							PivotElement					:= SEL(pPivotElement^[k] >= 97(*a*) AND_THEN pPivotElement^[k] <= 122(*z*), pPivotElement^[k], 	pPivotElement^[k] - 32);// a --> A
						END_IF
						// Find unequal char
						IF CompareElement <> PivotElement
							OR CompareElement = 0
							OR PivotElement = 0
						THEN
							EXIT;
						END_IF
					END_FOR
				UNTIL (CompareElement <= PivotElement) OR NOT (i < right)	END_REPEAT	
				REPEAT	
					j 										:= j-1;	
					pCmpElement								:= pCompareElement + (SizeOfStruct * TO_UDINT(j-1));
					FOR k := 0 TO MAX_WSTRING_LENGTH DO // Find unequal char
						// element 1,2 to upper char 	https://www.uni-due.de/hummell/infos/ascii/
						IF pCmpElement^[k] = 0 
							AND IgnoreBlank
						THEN
							CompareElement					:= 127;
						ELSE
							CompareElement					:= SEL(pCmpElement^[k] >= 97(*a*)	AND_THEN pCmpElement^[k] <= 122(*z*), 	pCmpElement^[k],pCmpElement^[k] - 32);		// a --> A
						END_IF
						IF pPivotElement^[k] = 0 
							AND IgnoreBlank
						THEN
							PivotElement					:= 127;
						ELSE
							PivotElement					:= SEL(pPivotElement^[k] >= 97(*a*) AND_THEN pPivotElement^[k] <= 122(*z*), pPivotElement^[k], 	pPivotElement^[k] - 32);// a --> A
						END_IF
						// Find unequal char
						IF CompareElement <> PivotElement
							OR CompareElement = 0
							OR PivotElement = 0
						THEN
							EXIT;
						END_IF
					END_FOR
				UNTIL (CompareElement >= PivotElement) OR NOT (j > left)	END_REPEAT		
			ELSE	// sort ascending
				REPEAT	
					i 										:= i+1;
					pCmpElement								:= pCompareElement + (SizeOfStruct * TO_UDINT(i-1));
					FOR k := 0 TO MAX_WSTRING_LENGTH DO // Find unequal char
						// element 1,2 to upper char 	https://www.uni-due.de/hummell/infos/ascii/
						IF pCmpElement^[k] = 0 
							AND IgnoreBlank
						THEN
							CompareElement					:= 127;
						ELSE
							CompareElement					:= SEL(pCmpElement^[k] >= 97(*a*)	AND_THEN pCmpElement^[k] <= 122(*z*), 	pCmpElement^[k],pCmpElement^[k] - 32);		// a --> A
						END_IF
						IF pPivotElement^[k] = 0 
							AND IgnoreBlank
						THEN
							PivotElement					:= 127;
						ELSE
							PivotElement					:= SEL(pPivotElement^[k] >= 97(*a*) AND_THEN pPivotElement^[k] <= 122(*z*), pPivotElement^[k], 	pPivotElement^[k] - 32);// a --> A
						END_IF
						// Find unequal char
						IF CompareElement <> PivotElement
							OR CompareElement = 0
							OR PivotElement = 0
						THEN
							EXIT;
						END_IF
					END_FOR
				UNTIL (CompareElement >= PivotElement)	OR NOT (i < right)	END_REPEAT;				
				REPEAT	
					j 										:= j-1;	
					pCmpElement								:= pCompareElement + (SizeOfStruct * TO_UDINT(j-1));
					FOR k := 0 TO MAX_WSTRING_LENGTH DO // Find unequal char
						// element 1,2 to upper char 	https://www.uni-due.de/hummell/infos/ascii/
						IF pCmpElement^[k] = 0 
							AND IgnoreBlank
						THEN
							CompareElement					:= 127;
						ELSE
							CompareElement					:= SEL(pCmpElement^[k] >= 97(*a*)	AND_THEN pCmpElement^[k] <= 122(*z*), 	pCmpElement^[k],pCmpElement^[k] - 32);		// a --> A
						END_IF
						IF pPivotElement^[k] = 0 
							AND IgnoreBlank
						THEN
							PivotElement					:= 127;
						ELSE
							PivotElement					:= SEL(pPivotElement^[k] >= 97(*a*) AND_THEN pPivotElement^[k] <= 122(*z*), pPivotElement^[k], 	pPivotElement^[k] - 32);// a --> A
						END_IF
						// Find unequal char
						IF CompareElement <> PivotElement
							OR CompareElement = 0
							OR PivotElement = 0
						THEN
							EXIT;
						END_IF
					END_FOR
				UNTIL (CompareElement <= PivotElement) OR NOT (j > left)	END_REPEAT;
			END_IF
			IF i >= j THEN
				endSubLoop									:= TRUE;
			ELSE                    					
				Allocate(SizeOfStruct);
				pElement_1									:= pData + (SizeOfStruct * TO_UDINT(j-1));
				pElement_2									:= pData + (SizeOfStruct * TO_UDINT(i-1));
				
				IF pElement_Tmp = 0 
					OR_ELSE MEMCPY(pElement_Tmp, pElement_1,	SizeOfStruct) = 0
					OR_ELSE MEMCPY(pElement_1,	pElement_2,		SizeOfStruct) = 0
					OR_ELSE MEMCPY(pElement_2,	pElement_Tmp,	SizeOfStruct) = 0
				THEN
					byWSTRING								:= FALSE;
					RETURN;	
				END_IF

			END_IF
		UNTIL endSubLoop END_REPEAT;		
		stack[stackCount] 									:= TO_UDINT(right); 	// save right in stack			
		IF stackCount < 32              					
		THEN                            					
			stackCount 										:= stackCount +1;
		ELSE															// Error stack Limit    
			endMainLoop 									:= TRUE;
			byWSTRING										:= FALSE;			
		END_IF                          					
		right 												:= MAX(left, i-1);
	ELSE                                
		IF stackCount = 1 THEN          
			endMainLoop 									:= TRUE;
		ELSE                            					
			left 											:= right+1;       
			stackCount 										:= stackCount -1;	// load from stack
			right											:= TO_DINT(stack[stackCount]);
		END_IF
	END_IF
END_WHILE
END_METHOD

METHOD FB_exit : BOOL
VAR_INPUT
	bInCopyCode : BOOL; // if TRUE, the exit method is called for exiting an instance that is copied afterwards (online change).
END_VAR
IF NOT bInCopyCode AND pElement_Tmp <> 0
THEN //Release memory in case the PLC stopps
	__DELETE(pElement_Tmp);
END_IF
END_METHOD

END_FUNCTION_BLOCK

// POUs/EventLogger/ReadEvents/EventlogRead
{attribute 'no_check'}
//Read TwinCat ADS evenlogger messages via ADS into PLC in Unicode format
FUNCTION_BLOCK EventlogRead EXTENDS FbBase
VAR CONSTANT
	IGRP_ENUMEVENTS											: UDINT := 16#190;
	IOFFS_ENUM_CONTINUE										: UDINT := 16#1020;
	IOFFS_ENUM_CLOSE										: UDINT := 16#1030;
                                        					
	IGRP_GETTEXT											: UDINT := 16#1F4;
	IOFFS_GETCOMPLETESTRING									: UDINT := 16#0;
	IOFFS_GETSOURCENAME										: UDINT := 16#1;
                                        					
	IOFFS_BEGINENUMACTIVE									: UDINT := 16#0;
	IOFFS_BEGINENUMLOGGED									: UDINT := 16#1;
                                        	
	IGRP_TCEVENTSTREAM_SIMPLE								: UDINT := 16#1;
	IOFFS_TCEVENTCLASS_NONE 								: UDINT := 16#0;
END_VAR
VAR_OUTPUT CONSTANT
	MIN_EVENT												: INT := 1; 
	MAX_EVENT												: INT := PARAM.EVENT_HANDLING_CONFIG.EVENTLOG_READ_MAX_EVENTS ; //End index event list  - see library parameter to customize parameter
	
{attribute 'displaymode':='binary'}
	OPTION_USE_STATE_FOR_TIMESTAMP							: 	BYTE :=2#0000_0001; //option to enable timestamp according to event state instead of only signaled timestamp
{attribute 'displaymode':='binary'}
	OPTION_GET_HOSTNAME_FOR_EACH_EVENT						: 	BYTE :=2#0000_0010; //option to read host name for each single event
END_VAR                                 					
VAR_INPUT                               					
	LangId													: eLCID := eLCID.US; //See LCID 	
	NetId													: T_AMSNetId := '';
	TimeOut													: TIME := DEFAULT_ADS_TIMEOUT;
	TimezoneBias											: DINT; //Timezone bias to UTC in minutes - As timestamp provided by Evetlogger is in UTC
{attribute 'displaymode':='binary'}
	Options													: BYTE := 2#0000_0000; 
END_VAR                                 					
VAR_OUTPUT                              					
	Event													: ARRAY [MIN_EVENT..MAX_EVENT] OF EVENTLOG_READ_DATA; //Event list 
	TotalNumberOfEvents										: INT := 0; //Number of events in list
	QuitReqNumberOfEvents									: INT := 0; //Number of events in list where quit is required
	CurrentEventCount										: INT := 0; //Count down the number of events need to read 
	ExecutionTime											: TIME; //Total cycle time to read all events
	ClassStatus												: DWORD; //Overview of active TC event classes - bit number is equivalent to TcEventClass count
END_VAR
VAR
(* Local memory ********************************************)
	MemLastErrorId											:	UDINT;
	MemTargetNetId											: T_AMSNetId;
	ReadBytes												: UDINT;
	MemTimeStartCycle										: TIME;
	MemClassStatus											: DWORD;
	MemEventFiletime										: T_FILETIME;	                         					
	MemADSEvent												: EVENTLOG_READ_DATA;
	                                    					
	EventStream												: EVENTLOG_READ_STREAM;
	HandleInfo												: EVENTLOG_READ_HANDLEINFO;
	PassHandleInfo											: EVENTLOG_READ_HANDLEINFO;

	CopyLen													:	UDINT;
(* Timer *******************************************************)

(* Trigger *****************************************************)
	
(* function-blocks *********************************************)
	fbAdsRead												: ADSREAD;
	fbAdsReadWrite											: ADSRDWRTEX;
	fbAdsWrite												: ADSWRITE;
	fbGetHostName											: FB_GetHostName;
	
(* Error *******************************************************)

(* internal used dummys *************************************)
	i														: 	UINT := 0 ;
END_VAR

	(* Read Eventlogger messages via ADS into the PLC  			 Unicode	*)
	(************************************************************************)

(* action **************************************************************************)
rtExecute(CLK := Execute);
CASE State OF
	0: 	(* Begin *)
		IF rtExecute.Q
		THEN
			Busy 											:= TRUE;
			Done 											:= FALSE;
			Error 											:= FALSE;
			ErrorId 										:= 0;
			fbAdsRead(READ := FALSE);           			
			fbAdsReadWrite(WRTRD := FALSE);     			
			fbAdsWrite(WRITE := FALSE);         			
			fbGetHostName(bExecute := FALSE);   			
			MemTimeStartCycle								:= TIME();
			MemClassStatus									:= 0;
			State 											:= 1;
                                                				
		ELSIF NOT Execute                       				
		THEN                                    				
			Done											:= FALSE;
			Busy 											:= FALSE;
			Error 											:= FALSE;
			ErrorId 										:= 0;
		END_IF

	1:	(* Get Handle*)
		fbAdsRead(
			NETID		:= NetId,
			PORT		:= AMSPORT_EVENTLOG,
			IDXGRP		:= IGRP_ENUMEVENTS,
			IDXOFFS		:= 16#1000 + IOFFS_BEGINENUMACTIVE,
			LEN			:= SIZEOF(HandleInfo),
			DESTADDR	:= ADR(HandleInfo),
			READ		:= TRUE,
			TMOUT		:= Timeout,
			BUSY		=> ,
			ERR			=> ,
			ErrId		=> );

		IF NOT fbAdsRead.BUSY
		THEN
			IF NOT fbAdsRead.ERR
			THEN
				CurrentEventCount 							:= LIMIT(0,DWORD_TO_INT(HandleInfo.Count),MAX_EVENT);
				TotalNumberOfEvents 						:= CurrentEventCount;
				QuitReqNumberOfEvents						:= CurrentEventCount;
				
				IF CurrentEventCount < 1
				THEN (* no actice event *)
					MEMSET(ADR(Event),0,SIZEOF (Event)); (* alle Events loeschen *)
					state 									:= 99;
				ELSE (* start reading data - deleting rest of current list *)
					MEMSET(ADR(Event[MIN(TotalNumberOfEvents + 1,MAX_EVENT)]),0, SIZEOF(Event[1]) * TO_UDINT((MAX_EVENT - TotalNumberOfEvents)));
					
					state 									:= 2;
				END_IF
				
			ELSE
				CurrentEventCount 							:= 1;
				TotalNumberOfEvents 						:= 1;
				QuitReqNumberOfEvents						:= 1;				
				ErrorId										:= fbAdsRead.ERRID;
				MEMSET(ADR(Event),0,SIZEOF (Event)); (* alle Events loeschen *)
				Event[1].eClass								:= TCEVENTCLASS_ALARM;
				Event[1].MsgText							:= WCONCAT("Error get event handle - Error ID: ", TO_WSTRING(ErrorId));
				Event[1].MegLen								:= TO_DWORD(WLEN(Event[1].MsgText));
				Event[1].Source								:= "<Unknown>";	
				Event[1].Computer							:= '<Local>';	
				
				State 										:= 99;
			END_IF
			fbAdsRead(READ := FALSE);		
		END_IF

	(* Read Event Stream **************************************************************)
	2: 
		PassHandleInfo.Enum 								:= HandleInfo.Enum;
		PassHandleInfo.Count 								:= 1;

		fbAdsReadWrite(
			NETID		:= NetId,
			PORT		:= AMSPORT_EVENTLOG,
			IDXGRP		:= IGRP_ENUMEVENTS,
			IDXOFFS		:= IOFFS_ENUM_CONTINUE,
			WRITELEN	:= SIZEOF(PassHandleInfo),
			READLEN		:= SIZEOF(EventStream),
			SRCADDR		:= ADR(PassHandleInfo),
			DESTADDR	:= ADR(EventStream),
			WRTRD		:= TRUE,
			TMOUT		:= Timeout,
			BUSY		=> ,
			ERR			=> ,
			ErrId		=> ,
			COUNT_R		=> ReadBytes);
			
		IF NOT fbAdsReadWrite.BUSY
		THEN
			IF NOT fbAdsReadWrite.ERR
			THEN
				IF EventStream.data.zFmtProgId = '' THEN
					EventStream.data.zFmtProgId 			:= 'TcEventFormatter.TcXmlFormatter';
				END_IF
				EventStream.cbStream 						:= EventStream.cbStream + 2;
				EventStream.count 							:= TO_DWORD(LangId);
				(* Target NetId from Event array *)
				MemTargetNetId 								:= F_CreateAmsNetId(EventStream.data.AdsAddr);
				
				MEMSET(ADR(MemAdsEvent),0,SIZEOF(MemAdsEvent));
					
				MemADSEvent.eClass							:= DWORD_TO_UINT(EventStream.data.Class);
				MemADSEvent.id 								:= EventStream.data.Id;
				MemADSEvent.SourceId						:= EventStream.data.SrcId;
				MemADSEvent.State							:= EventStream.data.State;
				MemADSEvent.Flags							:= EventStream.data.Flags;
						
				IF NOT Options.0
				THEN
					MemADSEvent.Timestamp					:= FILETIME_TO_DCTIME64(EventStream.data.TimeSignaled);							
				ELSE
					CASE MemADSEvent.State OF
					TCEVENTSTATE_SIGNALED:	
						MemADSEvent.Timestamp				:= FILETIME_TO_DCTIME64(EventStream.data.TimeSignaled);							
					TCEVENTSTATE_RESET:									
						MemADSEvent.Timestamp				:= FILETIME_TO_DCTIME64(EventStream.data.TimeReseted);	
					TCEVENTSTATE_CONFIRMED:					
						MemADSEvent.Timestamp				:= FILETIME_TO_DCTIME64(EventStream.data.TimeConfirmed);	
					TCEVENTSTATE_RESETCON:			
						MemADSEvent.Timestamp				:= MAX(FILETIME_TO_DCTIME64(EventStream.data.TimeReseted),FILETIME_TO_DCTIME64(EventStream.data.TimeConfirmed));				
					ELSE //TCEVENTSTATE_INVALID:
						MemADSEvent.Timestamp				:= FILETIME_TO_DCTIME64(EventStream.data.TimeSignaled);	
					END_CASE					
				END_IF
				IF TimezoneBias > 0
				THEN
					MemADSEvent.Timestamp					:= MemADSEvent.Timestamp + (60 * EC_DCTIME_TICKSPERSEC64 * TO_ULINT(TimezoneBias));
				ELSIF TimezoneBias < 0
				THEN
					MemADSEvent.Timestamp					:=  MemADSEvent.Timestamp - (TO_ULINT(ABS(TimezoneBias)) * 60 * EC_DCTIME_TICKSPERSEC64);
				END_IF
				MemADSEvent.TimestampDT						:= FILETIME_TO_DT(DCTIME64_TO_FILETIME(MemADSEvent.Timestamp));	
				MemClassStatus								:= SETBIT32(MemClassStatus, UINT_TO_SINT(Event[CurrentEventCount].eClass));
				state 										:= 3;
			ELSE
				ErrorId 									:= fbAdsReadWrite.ErrId;
				MEMSET(ADR(MemTargetNetId),0,SIZEOF(MemTargetNetId));
				MEMSET(ADR(MemAdsEvent),0,SIZEOF(MemAdsEvent));	
				MemADSEvent.eClass							:= TCEVENTCLASS_ALARM;				
				MemADsEvent.MsgText							:= WCONCAT("Error read event stream - Error ID: ", TO_WSTRING(ErrorId));
				MemADsEvent.MegLen							:= TO_DWORD(WLEN(MemADsEvent.MsgText));
				EventStream.count 							:= TO_DWORD(LangId);
				MemClassStatus								:= SETBIT32(MemClassStatus, UINT_TO_SINT(Event[CurrentEventCount].eClass));
				state 										:= 4;				
			END_IF
			
			fbAdsReadWrite(WRTRD := FALSE);		

		END_IF

	3:	(* Read Msg Text *)
		fbAdsReadWrite(
			NETID		:= NetId,
			PORT		:= AMSPORT_EVENTLOG,
			IDXGRP		:= IGRP_GETTEXT,
			IDXOFFS		:= IOFFS_GETCOMPLETESTRING,
			WRITELEN	:= EventStream.cbStream ,
			READLEN		:= SIZEOF(EventStream.data.evtData.Temp),
			SRCADDR		:= ADR(EventStream),
			DESTADDR	:= ADR(EventStream.data.evtData.Temp),
			WRTRD		:= TRUE,
			TMOUT		:= Timeout,
			BUSY		=> ,
			ERR			=> ,
			ErrId		=> ,
			COUNT_R		=> ReadBytes);

		IF NOT fbAdsReadWrite.BUSY
		THEN
			IF NOT fbAdsReadWrite.ERR
			THEN
				//Use unicode
				CopyLen										:= MIN(ReadBytes, SIZEOF(MemADsEvent.MsgText) - 2);
				MEMCPY(ADR(MemADsEvent.MsgText),ADR(EventStream.data.evtData.Temp),CopyLen);
				MemADsEvent.MegLen							:= CopyLen;
				MemADsEvent.MsgText[CopyLen]				:= 0; 
				
				state 										:= 4;
			ELSE
				ErrorId 									:= fbAdsReadWrite.ErrId;
				MemADsEvent.MsgText							:= WCONCAT("Error read event message - Error ID: ", TO_WSTRING(ErrorId));
				MemADsEvent.MegLen							:= TO_DWORD(WLEN(MemADsEvent.MsgText));
				State 										:= 4;
			END_IF
			fbAdsReadWrite(WRTRD := FALSE);		

		END_IF

	4:	(* Read Source Name *)
		PassHandleInfo.Enum 								:= HandleInfo.Enum;
		PassHandleInfo.Count 								:= 1;

		fbAdsReadWrite(
			NETID		:= NetId,
			PORT		:= AMSPORT_EVENTLOG,
			IDXGRP		:= IGRP_GETTEXT,
			IDXOFFS		:= IOFFS_GETSOURCENAME,
			WRITELEN	:= EventStream.cbStream,
			READLEN		:= SIZEOF(EventStream.data.evtData.Temp),
			SRCADDR		:= ADR(EventStream),
			DESTADDR	:= ADR(EventStream.data.evtData.Temp),
			WRTRD		:= TRUE,
			TMOUT		:= Timeout,
			BUSY		=> ,
			ERR			=> ,
			ErrId		=> ,
			COUNT_R		=> ReadBytes);

		IF NOT fbAdsReadWrite.BUSY
		THEN
			IF NOT fbAdsReadWrite.ERR
			THEN
				CopyLen										:= MIN(ReadBytes, SIZEOF(MemADsEvent.Source) - 2);
				MEMCPY(ADR(MemADsEvent.Source),ADR(EventStream.data.evtData.Temp),CopyLen);						
		
			ELSIF fbAdsReadWrite.ErrId = 16#80070057 OR  fbAdsReadWrite.ErrId = 16#80030002
			THEN
				MemAdsEvent.Source							:= WCONCAT("Name unknown id ", TO_WSTRING(EventStream.data.SrcId));
			ELSE
				ErrorId 									:= fbAdsReadWrite.ErrId;
				MemAdsEvent.Source				 			:= "<Unknown>";
			END_IF
		
			state											:= 5;
			fbAdsReadWrite(WRTRD := FALSE);		

		END_IF
		
	5: (* Read Host Name *)
		fbGetHostName(
			sNetID		:= MemTargetNetId ,
			bExecute	:= fbGetHostName.sHostName <> '' OR Options.1,
			tTimeout	:= Timeout,
			bBusy		=> ,
			bError		=> ,
			nErrId		=> ,
			sHostName	=> );

		IF NOT fbGetHostName.bBusy
		THEN
			IF fbGetHostName.bError
			THEN
				MemAdsEvent.Computer						:= '<Unknown>';
			ELSE
				MemAdsEvent.Computer						:= fbGetHostName.sHostName;		
			END_IF

			//Copy event to 
			Event[CurrentEventCount]						:= MemAdsEvent;	
	
			//Count quit required events 
			IF NOT MemAdsEvent.Flags.1
			THEN
				QuitReqNumberOfEvents						:= QuitReqNumberOfEvents - 1;
			END_IF
					
			(* other messages *)
			CurrentEventCount 								:= CurrentEventCount - 1;
			IF CurrentEventCount < 1 THEN
				state 										:= 99;
			ELSE
				state 										:= 2;
			END_IF
			
			fbGetHostName(bExecute := FALSE);
		END_IF

	99: 	(* Close *)				
		fbAdsWrite(
			NETID	:= NetId,
			PORT	:= AMSPORT_EVENTLOG,
			IDXGRP	:= IGRP_ENUMEVENTS,
			IDXOFFS	:= IOFFS_ENUM_CLOSE,
			LEN		:= SIZEOF(HandleInfo.Enum),
			SRCADDR	:= ADR(HandleInfo),
			WRITE	:= state = 99,
			TMOUT	:= Timeout,
			BUSY	=> ,
			ERR		=> ,
			ErrId	=> );

		IF NOT fbAdsWrite.BUSY
		THEN
			ExecutionTime	 								:= TIME() - MemTimeStartCycle;
			Done											:= ErrorId = 0 AND Busy;
			Error 											:= NOT Done;
			ErrorId 										:= SEL(fbAdsWrite.ERR, ErrorId,fbAdsWrite.ErrId);
			MemLastErrorid									:= ErrorId;
			ClassStatus										:= MemClassStatus;
			Busy 											:= FALSE;
			State 											:= 0;

			fbAdsWrite(WRITE := FALSE);
		END_IF

	END_CASE
	
(*************************************************************************************************)

PROPERTY PUBLIC optGetHostNameForEachEvent : bool
GET
optGetHostNameForEachEvent := Options.1;
END_GET
SET
Options.1 := optGetHostNameForEachEvent;
END_SET
END_PROPERTY

PROPERTY PUBLIC optUseStateForTimestamp : bool
GET
optUseStateForTimestamp := Options.0;
END_GET
SET
Options.0 := optUseStateForTimestamp;
END_SET
END_PROPERTY

END_FUNCTION_BLOCK

// POUs/EventLogger/TriggerEvents/EventHandling
{attribute 'no_check'}
//ADSLOGEVENT wrapper for a convenient and pre configured use - see Beckhoff documentation for more information about AdsEventLogger
//See Param constanst to configure whether the TcEventClass need to be acknowledged (confirmation required) 
FUNCTION_BLOCK EventHandling
VAR_INPUT
	Flag													:	BOOL := FALSE; //Fire event 
	ConfirmTrig												:	BOOL := FALSE; //Ack event
	MsgId													:	UINT := 0; //Event number
	SourceId												: 	UDINT:= 0; //Event source number
	eClass													:	E_TcEventClass := TCEVENTCLASS_ALARM; (*	TC2_SYSTEM.TCEVENTCLASS_NONE		
																											TC2_SYSTEM.TCEVENTCLASS_MAINTENANCE
																											TC2_SYSTEM.TCEVENTCLASS_MESSAGE		
																											TC2_SYSTEM.TCEVENTCLASS_HINT		
																											TC2_SYSTEM.TCEVENTCLASS_STATEINFO	
																											TC2_SYSTEM.TCEVENTCLASS_INSTRUCTION	
																											TC2_SYSTEM.TCEVENTCLASS_WARNING		
																											TC2_SYSTEM.TCEVENTCLASS_ALARM		
																											TC2_SYSTEM.TCEVENTCLASS_PARAMERROR	*)

	Text1													:	STRING(20) := ''; //Short info text with lenght 20 chars 
	Text2													:	STRING(40) := ''; //Long info text with lenght 40 chars
	pText3													:	POINTER TO STRING := 0; //Pointer to extended info text 
END_VAR
VAR_OUTPUT
{attribute 'displaymode':='hex'}
	State													:	UDINT ; (*	TCEVENTSTATE_INVALID  	: WORD := 16#0000; 		
																			TCEVENTSTATE_SIGNALED  	: WORD := 16#0001; 		- The event is signaled 
																			TCEVENTSTATE_RESET  	: WORD := 16#0002; 		- The event is gone 
																			TCEVENTSTATE_CONFIRMED  : WORD := 16#0010 (16); - The event is confirmed 
																			TCEVENTSTATE_RESETCON  	: WORD := 16#0012 (18); - The event is gone AND confirmed *)
{attribute 'displaymode':='binary'}
	Status													:	DWORD; (*	.0 - .8 = event <class id>  / .15 confirm required / .16 = Level 0 , .17 = Level 1 , .18 = Level 2, .......... / .31 active
																			TCEVENTCLASS_NONE			:=0,
																			TCEVENTCLASS_MAINTENANCE	:=1,
																			TCEVENTCLASS_MESSAGE		:=2,
																			TCEVENTCLASS_HINT			:=3,
																			TCEVENTCLASS_STATEINFO		:=4, 
																			TCEVENTCLASS_INSTRUCTION	:=5,
																			TCEVENTCLASS_WARNING		:=6,
																			TCEVENTCLASS_ALARM			:=7,
																			TCEVENTCLASS_PARAMERROR		:=8	 *)
END_VAR
VAR
	format													:	STRING(6) := '%s%s%s';
	pPara													:	ARRAY[1..3] OF POINTER TO BYTE;
	TmpString												:	STRING(1) := '';
	AdsEvent												:	ADSLOGEVENT :=(
																	NETID				:= '',
																	PORT				:= AMSPORT_EVENTLOG,
																	TMOUT 				:= DEFAULT_ADS_TIMEOUT,
																	EventDataLength		:= 0,	
																	EventConfigData 	:= (
																		Class 				:= TCEVENTCLASS_ALARM,
																		Prio 				:= TCEVENTPRIO_IMPLICIT,
																		ProgId 				:= 'TcEventFormatter.TcXmlFormatter',
																		Flags 				:= TCEVENTFLAG_LOG OR TCEVENTFLAG_SRCID, // 16#0140 (* T *),
																		StreamType 			:= TCEVENTSTREAM_SIMPLE (* TCEVENTSTREAM_NORMAL *),
																		bQuitRequired 		:= TRUE));
END_VAR

(* EventHandling including textinfos which are send to the eventlogger  	v4.3	*)
(* specific eventclasses have to be quit, see Param.EventConfig...					*)
(************************************************************************************)

(* sequence *************************************************************)
	IF Status.31 //Message active
	THEN (* work EventLogger *)
		AdsEvent(
			NETID			:= ,(* see declaration *)
			PORT			:= ,(* see declaration *)
			Event			:= NOT AdsEvent.FbCleanup AND(Flag OR AdsEvent.EventState = TCEVENTSTATE_INVALID AND NOT AdsEvent.Quit), (* Set Event until state <> invalid *)
			EventQuit		:= AdsEvent.EventState <> TCEVENTSTATE_INVALID
								AND AdsEvent.EventConfigData.bQuitRequired
								AND NOT AdsEvent.Eventstate.4 //confirmed
								AND NOT AdsEvent.Quit
								AND(
								ConfirmTrig
								OR AdsEvent.EventQuit), (* quit send *)
			EventConfigData	:= ,(* see declaration *)
			EventDataAddress:= ADR(pPara),
			EventDataLength	:= ,(* see declaration *)
			FbCleanup		:= NOT AdsEvent.FbCleanup AND(AdsEvent.Err OR AdsEvent.EventState = TCEVENTSTATE_RESETCON),
			TMOUT			:= ,(* see declaration *)
			EventState		=> ,
			Err				=> ,
			ErrId			=> ,
			Quit			=> );
			
		IF AdsEvent.Event 
			AND AdsEvent.EventState = TCEVENTSTATE_INVALID
		THEN
			State 											:= SEL(Flag, TCEVENTSTATE_RESET, TCEVENTSTATE_SIGNALED);
		ELSIF AdsEvent.Quit
			AND AdsEvent.EventState = TCEVENTSTATE_INVALID
			AND AdsEvent.EventQuit
			OR 
			AdsEvent.FbCleanup		
		THEN
			State 											:= TCEVENTSTATE_RESETCON;
		ELSIF(AdsEvent.Err OR NOT AdsEvent.Event AND AdsEvent.EventState = TCEVENTSTATE_INVALID)
			AND_THEN Gvl.EventHandlingStatistic.CountOut(Status)
		THEN
			State											:= TCEVENTSTATE_INVALID;
		ELSE
			State											:= MAX(State, AdsEvent.EventState);
		END_IF
			
	ELSIF Flag AND SourceId > 0 
	THEN (* fire event *)
		IF PARAM.EVENT_HANDLING_CONFIG.ENABLE_DYNAMIC_EVENT_MSG_FORMAT
		THEN
			IF pText3 <> 0 AND_THEN pText3^[0] > 0
			THEN 
				format 										:= '%s%s%s'; 
			ELSIF Text2[0] > 0 
			THEN 
				format 										:= '%s%s';
			ELSIF Text1[0] > 0 
			THEN 												
				format 										:= '%s';
			ELSE
				format 										:= '';
			END_IF
		END_IF
							 
		AdsEvent.EventConfigData.DataFormatStrAddress		:= ADR(format);
		AdsEvent.EventConfigData.Id 						:= UINT_TO_UDINT(MsgID);
		AdsEvent.EventConfigData.SourceId 					:= SourceId;
		Status												:= Gvl.EventHandlingStatistic.InitEvent(SetClass := eClass, EventConfig := AdsEvent.EventConfigData);		

		(* Data *)
		pPara[1] 											:= ADR(Text1);
		pPara[2] 											:= ADR(Text2);
		pPara[3] 											:= SEL(pText3 <> 0,ADR(TmpString) ,pText3);
	
		IF AdsEvent.Err AND NOT AdsEvent.FbCleanup
		THEN
			AdsEvent(
				Event			:= FALSE,
				EventQuit 		:= FALSE,
				EventDataAddress:= ADR(pPara),
				FbCleanup		:= TRUE,
				EventState		=> );
				
		ELSE (* Fire Event *)
			AdsEvent( 	
				Event			:= FALSE,
				EventQuit 		:= FALSE, 
				FbCleanup 		:= FALSE, 
				EventDataAddress:= ADR(pPara));
						
			AdsEvent( 	Event 	:= TRUE);
			IF NOT AdsEvent.Err AND_THEN Gvl.EventHandlingStatistic.CountIn(Status) //Add event to statistic and continue if added successfully
			THEN			
				State 										:= TCEVENTSTATE_SIGNALED;
			END_IF
						
		END_IF
	END_IF

(**********************************************************************************)

END_FUNCTION_BLOCK

// POUs/EventLogger/TriggerEvents/EventHandlingConfirmIsReq
{attribute 'no_check'}
//Returns status of "QuitRequired" configuration for corresponding event class (see library Param) 
FUNCTION EventHandlingConfirmIsReq : BOOL
VAR_INPUT
	TcEventClass											:	E_TcEventClass;
END_VAR
VAR
END_VAR

	CASE tcEventClass OF
	Tc2_System.TCEVENTCLASS_NONE:			EventHandlingConfirmIsReq	:= PARAM.EVENT_HANDLING_CONFIG.CLASS_NONE_QUIT_REQUIRED;	
	Tc2_System.TCEVENTCLASS_MAINTENANCE:	EventHandlingConfirmIsReq	:= PARAM.EVENT_HANDLING_CONFIG.CLASS_MAINTENANCE_QUIT_REQUIRED;		
	Tc2_System.TCEVENTCLASS_MESSAGE:		EventHandlingConfirmIsReq	:= PARAM.EVENT_HANDLING_CONFIG.CLASS_MESSAGE_QUIT_REQUIRED;			
	Tc2_System.TCEVENTCLASS_HINT:			EventHandlingConfirmIsReq	:= PARAM.EVENT_HANDLING_CONFIG.CLASS_HINT_QUIT_REQUIRED;	
	Tc2_System.TCEVENTCLASS_STATEINFO:		EventHandlingConfirmIsReq	:= PARAM.EVENT_HANDLING_CONFIG.CLASS_STATEINFO_QUIT_REQUIRED;	
	Tc2_System.TCEVENTCLASS_INSTRUCTION:	EventHandlingConfirmIsReq	:= PARAM.EVENT_HANDLING_CONFIG.CLASS_INSTRUCTION_QUIT_REQUIRED;	
	Tc2_System.TCEVENTCLASS_WARNING:		EventHandlingConfirmIsReq	:= PARAM.EVENT_HANDLING_CONFIG.CLASS_WARNING_QUIT_REQUIRED;	
	Tc2_System.TCEVENTCLASS_ALARM:			EventHandlingConfirmIsReq	:= PARAM.EVENT_HANDLING_CONFIG.CLASS_ALARM_QUIT_REQUIRED;	
	Tc2_System.TCEVENTCLASS_PARAMERROR:		EventHandlingConfirmIsReq	:= PARAM.EVENT_HANDLING_CONFIG.CLASS_PARAMERROR_QUIT_REQUIRED;		
	ELSE                                                    
		EventHandlingConfirmIsReq										:= PARAM.EVENT_HANDLING_CONFIG.CLASS_ALARM_QUIT_REQUIRED;
	END_CASE

END_FUNCTION

// POUs/EventLogger/TriggerEvents/EventHandlingGrp10
{attribute 'no_check'}
//Event group with single source id - for a convenient control of <MAX_EVENTS>
//Each single event handling FB is accessible, so that signal flag, information text and alarm class could be used
FUNCTION_BLOCK EventHandlingGrp10
VAR_OUTPUT CONSTANT
	MIN_EVENT												:	INT := 1; 
	MAX_EVENT												:	INT := 10;
END_VAR                                                 	
VAR_INPUT                                               	
	ConfirmTrig												:	BOOL := FALSE; //Acknowledge event
	SourceId												: 	UDINT := 0; //Source id for all events of this group
	no														:	ARRAY [MIN_EVENT..MAX_EVENT] OF EventHandling; //Array of single event handling FBs 
	Disable													:	BOOL := FALSE; //Disable all events 
	AutoConfirm												:	BOOL := FALSE; //All events will be acknowledged if flag is gone *)
	SetClass												:	E_TcEventClass := TC2_SYSTEM.TCEVENTCLASS_ALARM;// if set class is <> ALARM -> all events set to this Eventclass
	MsgOffset												:	INT := 0; //Offset to change default message id to MIN_EVENT to MsgOffset
END_VAR                                                 	
VAR_OUTPUT    
{attribute 'displaymode':='binary'}
	Status													:	DWORD; (*	.0 - .8 = event of <class id> is active / .15 confirm required / .16 = Level 0 , .17 = Level 1 , .18 = Level 2, ..........
																			TCEVENTCLASS_NONE			:=0,	(* No class *)
																			TCEVENTCLASS_MAINTENANCE	:=1,	(* Maintenance hint *)
																			TCEVENTCLASS_MESSAGE		:=2,	(* Message *)
																			TCEVENTCLASS_HINT			:=3,	(* Hint *)
																			TCEVENTCLASS_STATEINFO		:=4,	(* State information *)
																			TCEVENTCLASS_INSTRUCTION	:=5,	(* Instruction *)
																			TCEVENTCLASS_WARNING		:=6,	(* Warning *)
																			TCEVENTCLASS_ALARM			:=7,	(* Alarm *)
																			TCEVENTCLASS_PARAMERROR		:=8		(* Parameter error *)  *)
	NoOfActiveEvents										:	INT;
END_VAR                                                 	
VAR                                                     	
	_Mem													:	BYTE;
	Disabled												:	BOOL;
	i 														:	INT;
END_VAR

(* EventHandlingGrp			V4.1	*)
(************************************)

(* status ***************************)
Status  													:= 0;
NoOfActiveEvents											:= 0;

IF(Disable OR SourceId = 0)AND Disabled
THEN
	RETURN;
ELSE	
	Disabled												:= Disable OR SourceId = 0;
	
	FOR i := MIN_EVENT TO MAX_EVENT 
	DO
		(* Init Default Class *)
		IF SetClass <> TC2_SYSTEM.TCEVENTCLASS_ALARM
			AND NOT _Mem.7
		THEN
			no[i].eClass										:= SetClass;
			_Mem.7											:= i = MAX_EVENT;
		END_IF                                  			
		                                        			
		IF Disable OR SourceId = 0              			
		THEN                                    			
			no[i].Flag 										:= FALSE;
			no[i].ConfirmTrig 								:= no[i].State <> TCEVENTSTATE_INVALID AND no[i].State <> TCEVENTSTATE_RESETCON;
		ELSIF ConfirmTrig                             			
		THEN                                    	
			no[i].ConfirmTrig 								:= TRUE;
			_Mem.0 											:= ConfirmTrig;
                                                			
		ELSIF _Mem.0                            			
		THEN                                    			
			no[i].ConfirmTrig 								:= FALSE;
			_Mem.0 											:= i <> MAX_EVENT;

		ELSIF AutoConfirm
		THEN
			IF NOT no[i].Flag
				AND no[i].State <> TCEVENTSTATE_INVALID
				AND no[i].State <> TCEVENTSTATE_RESETCON
			THEN
				no[i].ConfirmTrig 							:= TRUE;
			ELSE                                			
				no[i].ConfirmTrig 							:= FALSE;
			END_IF                              			
		END_IF                                  	
                                                	
		(* Mem current Event *)                 	
		IF no[i].State <> TCEVENTSTATE_INVALID OR no[i].Flag 
		THEN
			_Mem.1											:= TRUE;
			(* Call Event *)
			no[i](
				Flag	:= ,
				ConfirmTrig := ,
				MsgId	:= TO_UINT(i + MsgOffset),
				SourceId:= SourceId,
				eClass	:= (* see grp call *),
				Text1	:= (* see grp call *),
				Text2	:= (* see grp call *),
				pText3	:= (* see grp call *),
				State	=> );
		END_IF

		(* Set info flags *)
		IF	no[i].State <> TCEVENTSTATE_INVALID 
		THEN
			NoOfActiveEvents								:= NoOfActiveEvents + 1;
			Status											:= Status OR no[i].Status;
			Disabled										:= FALSE;
		ELSIF _Mem.1
		THEN (* Send one time info event is gone *)
			; 
		END_IF
	END_FOR	
END_IF
(*****************************************************************************************)

METHOD PUBLIC confirm : booL //Return value = TRUE if execution finished
VAR_INPUT
END_VAR
IF NoOfActiveEvents > 0
THEN
	FOR i := MIN_EVENT TO MAX_EVENT 
	DO
		no[i](ConfirmTrig := TRUE);
	END_FOR
	_Mem.0			:= TRUE;
END_IF

confirm		:= TRUE;
END_METHOD

PROPERTY PUBLIC confirmIsReq : BOOL
GET
confirmIsReq							:= Status.15;
END_GET
END_PROPERTY

PROPERTY PUBLIC isActive : BOOL
GET
IsActive 								:= Status <> 0;
END_GET
END_PROPERTY

END_FUNCTION_BLOCK

// POUs/EventLogger/TriggerEvents/EventHandlingGrp25
{attribute 'no_check'}
//Event group with single source id - for a convenient control of <MAX_EVENTS>
//Each single event handling FB is accessible, so that signal flag, information text and alarm class could be used
FUNCTION_BLOCK EventHandlingGrp25
VAR_OUTPUT CONSTANT
	MIN_EVENT												:	INT := 1; 
	MAX_EVENT												:	INT := 25;
END_VAR                                                 	
VAR_INPUT                                               	
	ConfirmTrig												:	BOOL := FALSE; //Acknowledge event
	SourceId												: 	UDINT := 0; //Source id for all events of this group
	no														:	ARRAY [MIN_EVENT..MAX_EVENT] OF EventHandling; //Array of single event handling FBs 
	Disable													:	BOOL := FALSE; //Disable all events 
	AutoConfirm												:	BOOL := FALSE; //All events will be acknowledged if flag is gone *)
	SetClass												:	E_TcEventClass := TC2_SYSTEM.TCEVENTCLASS_ALARM;// if set class is <> ALARM -> all events set to this Eventclass
	MsgOffset												:	INT := 0; //Offset to change default message id to MIN_EVENT to MsgOffset
END_VAR                                                 	
VAR_OUTPUT    
{attribute 'displaymode':='binary'}
	Status													:	DWORD; (*	.0 - .8 = event of <class id> is active / .15 confirm required / .16 = Level 0 , .17 = Level 1 , .18 = Level 2, ..........
																			TCEVENTCLASS_NONE			:=0,	(* No class *)
																			TCEVENTCLASS_MAINTENANCE	:=1,	(* Maintenance hint *)
																			TCEVENTCLASS_MESSAGE		:=2,	(* Message *)
																			TCEVENTCLASS_HINT			:=3,	(* Hint *)
																			TCEVENTCLASS_STATEINFO		:=4,	(* State information *)
																			TCEVENTCLASS_INSTRUCTION	:=5,	(* Instruction *)
																			TCEVENTCLASS_WARNING		:=6,	(* Warning *)
																			TCEVENTCLASS_ALARM			:=7,	(* Alarm *)
																			TCEVENTCLASS_PARAMERROR		:=8		(* Parameter error *)  *)
	NoOfActiveEvents										:	INT;																		
END_VAR                                                 	
VAR                                                     	
	_Mem													:	BYTE;
	Disabled												:	BOOL;
	i 														:	INT;
END_VAR

(* EventHandlingGrp			V4.1	*)
(************************************)

(* status ***************************)
Status  													:= 0;
NoOfActiveEvents											:= 0;

IF(Disable OR SourceId = 0)AND Disabled
THEN
	RETURN;
ELSE
	Disabled												:= Disable OR SourceId = 0;
	
	FOR i := MIN_EVENT TO MAX_EVENT 
	DO
		(* Init Default Class *)
		IF SetClass <> TC2_SYSTEM.TCEVENTCLASS_ALARM
			AND NOT _Mem.7
		THEN
			no[i].eClass										:= SetClass;
			_Mem.7											:= i = MAX_EVENT;
		END_IF                                  			
		                                        			
		IF Disable OR SourceId = 0              			
		THEN                                    			
			no[i].Flag 										:= FALSE;
			no[i].ConfirmTrig 								:= no[i].State <> TCEVENTSTATE_INVALID AND no[i].State <> TCEVENTSTATE_RESETCON;
		ELSIF ConfirmTrig                             			
		THEN                                    	
			no[i].ConfirmTrig 								:= TRUE;
			_Mem.0 											:= ConfirmTrig;
                                                			
		ELSIF _Mem.0                            			
		THEN                                    			
			no[i].ConfirmTrig 								:= FALSE;
			_Mem.0 											:= i <> MAX_EVENT;

		ELSIF AutoConfirm
		THEN
			IF NOT no[i].Flag
				AND no[i].State <> TCEVENTSTATE_INVALID
				AND no[i].State <> TCEVENTSTATE_RESETCON
			THEN
				no[i].ConfirmTrig 							:= TRUE;
			ELSE                                			
				no[i].ConfirmTrig 							:= FALSE;
			END_IF                              			
		END_IF                                  	
                                                	
		(* Mem current Event *)                 	
		IF no[i].State <> TCEVENTSTATE_INVALID OR no[i].Flag 
		THEN
			_Mem.1											:= TRUE;
			(* Call Event *)
			no[i](
				Flag	:= ,
				ConfirmTrig := ,
				MsgId	:= TO_UINT(i + MsgOffset),
				SourceId:= SourceId,
				eClass	:= (* see grp call *),
				Text1	:= (* see grp call *),
				Text2	:= (* see grp call *),
				pText3	:= (* see grp call *),
				State	=> );
		END_IF

		(* Set info flags *)
		IF	no[i].State <> TCEVENTSTATE_INVALID 
		THEN
			NoOfActiveEvents								:= NoOfActiveEvents + 1;
			Status											:= Status OR no[i].Status;
			Disabled										:= FALSE;
		ELSIF _Mem.1
		THEN (* Send one time info event is gone *)
			; 
		END_IF
	END_FOR	
END_IF
(*****************************************************************************************)

METHOD PUBLIC confirm : booL //Return value = TRUE if execution finished
VAR_INPUT
END_VAR
IF NoOfActiveEvents > 0
THEN
	FOR i := MIN_EVENT TO MAX_EVENT 
	DO
		no[i](ConfirmTrig := TRUE);
	END_FOR
	_Mem.0			:= TRUE;
END_IF

confirm		:= TRUE;
END_METHOD

PROPERTY PUBLIC confirmIsReq : BOOL
GET
confirmIsReq							:= Status.15;
END_GET
END_PROPERTY

PROPERTY PUBLIC isActive : BOOL
GET
IsActive 								:= Status <> 0;
END_GET
END_PROPERTY

END_FUNCTION_BLOCK

// POUs/EventLogger/TriggerEvents/EventHandlingGrp50
{attribute 'no_check'}
//Event group with single source id - for a convenient control of <MAX_EVENTS>
//Each single event handling FB is accessible, so that signal flag, information text and alarm class could be used
FUNCTION_BLOCK EventHandlingGrp50
VAR_OUTPUT CONSTANT
	MIN_EVENT												:	INT := 1; 
	MAX_EVENT												:	INT := 50;
END_VAR                                                 	
VAR_INPUT                                               	
	ConfirmTrig												:	BOOL := FALSE; //Acknowledge event
	SourceId												: 	UDINT := 0; //Source id for all events of this group
	no														:	ARRAY [MIN_EVENT..MAX_EVENT] OF EventHandling; //Array of single event handling FBs 
	Disable													:	BOOL := FALSE; //Disable all events 
	AutoConfirm												:	BOOL := FALSE; //All events will be acknowledged if flag is gone *)
	SetClass												:	E_TcEventClass := TC2_SYSTEM.TCEVENTCLASS_ALARM;// if set class is <> ALARM -> all events set to this Eventclass
	MsgOffset												:	INT := 0; //Offset to change default message id to MIN_EVENT to MsgOffset
END_VAR                                                 	
VAR_OUTPUT    
{attribute 'displaymode':='binary'}
	Status													:	DWORD; (*	.0 - .8 = event of <class id> is active / .15 confirm required / .16 = Level 0 , .17 = Level 1 , .18 = Level 2, ..........
																			TCEVENTCLASS_NONE			:=0,	(* No class *)
																			TCEVENTCLASS_MAINTENANCE	:=1,	(* Maintenance hint *)
																			TCEVENTCLASS_MESSAGE		:=2,	(* Message *)
																			TCEVENTCLASS_HINT			:=3,	(* Hint *)
																			TCEVENTCLASS_STATEINFO		:=4,	(* State information *)
																			TCEVENTCLASS_INSTRUCTION	:=5,	(* Instruction *)
																			TCEVENTCLASS_WARNING		:=6,	(* Warning *)
																			TCEVENTCLASS_ALARM			:=7,	(* Alarm *)
																			TCEVENTCLASS_PARAMERROR		:=8		(* Parameter error *)  *)
	NoOfActiveEvents										:	INT;
END_VAR                                                 	
VAR                                                     	
	_Mem													:	BYTE;
	Disabled												:	BOOL;
	i 														:	INT;
END_VAR

(* EventHandlingGrp			V4.1	*)
(************************************)

(* status ***************************)
Status  													:= 0;
NoOfActiveEvents											:= 0;

IF(Disable OR SourceId = 0)AND Disabled
THEN
	RETURN;
ELSE
	Disabled												:= Disable OR SourceId = 0;
	
	FOR i := MIN_EVENT TO MAX_EVENT 
	DO
		(* Init Default Class *)
		IF SetClass <> TC2_SYSTEM.TCEVENTCLASS_ALARM
			AND NOT _Mem.7
		THEN
			no[i].eClass										:= SetClass;
			_Mem.7											:= i = MAX_EVENT;
		END_IF                                  			
		                                        			
		IF Disable OR SourceId = 0              			
		THEN                                    			
			no[i].Flag 										:= FALSE;
			no[i].ConfirmTrig 								:= no[i].State <> TCEVENTSTATE_INVALID AND no[i].State <> TCEVENTSTATE_RESETCON;
		ELSIF Confirmtrig                             			
		THEN                                    	
			no[i].ConfirmTrig 								:= TRUE;
			_Mem.0 											:= Confirmtrig;
                                                			
		ELSIF _Mem.0                            			
		THEN                                    			
			no[i].ConfirmTrig 								:= FALSE;
			_Mem.0 											:= i <> MAX_EVENT;

		ELSIF AutoConfirm
		THEN
			IF NOT no[i].Flag
				AND no[i].State <> TCEVENTSTATE_INVALID
				AND no[i].State <> TCEVENTSTATE_RESETCON
			THEN
				no[i].ConfirmTrig 							:= TRUE;
			ELSE                                			
				no[i].ConfirmTrig 							:= FALSE;
			END_IF                              			
		END_IF                                  	
                                                	
		(* Mem current Event *)                 	
		IF no[i].State <> TCEVENTSTATE_INVALID OR no[i].Flag 
		THEN
			_Mem.1											:= TRUE;
			(* Call Event *)
			no[i](
				Flag	:= ,
				ConfirmTrig := ,
				MsgId	:= TO_UINT(i + MsgOffset),
				SourceId:= SourceId,
				eClass	:= (* see grp call *),
				Text1	:= (* see grp call *),
				Text2	:= (* see grp call *),
				pText3	:= (* see grp call *),
				State	=> );
		END_IF

		(* Set info flags *)
		IF	no[i].State <> TCEVENTSTATE_INVALID 
		THEN
			NoOfActiveEvents								:= NoOfActiveEvents + 1;
			Status											:= Status OR no[i].Status;
			Disabled										:= FALSE;
		ELSIF _Mem.1
		THEN (* Send one time info event is gone *)
			; 
		END_IF
	END_FOR	
END_IF
(*****************************************************************************************)

METHOD PUBLIC confirm : booL  //Return value = TRUE if execution finished
VAR_INPUT
END_VAR
IF NoOfActiveEvents > 0
THEN
	FOR i := MIN_EVENT TO MAX_EVENT 
	DO
		no[i](ConfirmTrig := TRUE);
	END_FOR
	_Mem.0			:= TRUE;
END_IF

confirm		:= TRUE;
END_METHOD

PROPERTY PUBLIC confirmIsReq : BOOL
GET
confirmIsReq							:= Status.15;
END_GET
END_PROPERTY

PROPERTY PUBLIC isActive : BOOL
GET
IsActive 								:= Status <> 0;
END_GET
END_PROPERTY

END_FUNCTION_BLOCK

// POUs/EventLogger/TriggerEvents/EventHandlingGrpCustomized
{attribute 'no_check'}
//Event group with single source id - for a convenient control of <MAX_EVENTS>
//Each single event handling FB is accessible, so that signal flag, information text and alarm class could be used
FUNCTION_BLOCK EventHandlingGrpCustomized
VAR_OUTPUT CONSTANT
	MIN_EVENT												:	INT := 1; 
	MAX_EVENT												:	INT := PARAM.EVENT_HANDLING_CONFIG.GRP_CUSTOMISED_MAX_EVENT; //Start index no of events - see library parameter to customize parameter
END_VAR                                                 	
VAR_INPUT                                               	
	ConfirmTrig												:	BOOL := FALSE; //Acknowledge event
	SourceId												: 	UDINT := 0; //Source id for all events of this group
	no														:	ARRAY [MIN_EVENT..MAX_EVENT] OF EventHandling; //Array of single event handling FBs 
	Disable													:	BOOL := FALSE; //Disable all events 
	AutoConfirm												:	BOOL := FALSE; //All events will be acknowledged if flag is gone *)
	SetClass												:	E_TcEventClass := TC2_SYSTEM.TCEVENTCLASS_ALARM;// if set class is <> ALARM -> all events set to this Eventclass
	MsgOffset												:	INT := 0; //Offset to change default message id to MIN_EVENT to MsgOffset
END_VAR                                                 	
VAR_OUTPUT                                              	
{attribute 'displaymode':='binary'}
	Status													:	DWORD; (*	.0 - .8 = event of <class id> is active / .15 confirm required / .16 = Level 0 , .17 = Level 1 , .18 = Level 2, ..........
																			TCEVENTCLASS_NONE			:=0,	(* No class *)
																			TCEVENTCLASS_MAINTENANCE	:=1,	(* Maintenance hint *)
																			TCEVENTCLASS_MESSAGE		:=2,	(* Message *)
																			TCEVENTCLASS_HINT			:=3,	(* Hint *)
																			TCEVENTCLASS_STATEINFO		:=4,	(* State information *)
																			TCEVENTCLASS_INSTRUCTION	:=5,	(* Instruction *)
																			TCEVENTCLASS_WARNING		:=6,	(* Warning *)
																			TCEVENTCLASS_ALARM			:=7,	(* Alarm *)
																			TCEVENTCLASS_PARAMERROR		:=8		(* Parameter error *)  *)
	NoOfActiveEvents										:	INT;
END_VAR                                                 	
VAR                                                     	
	_Mem													:	BYTE;
	Disabled												:	BOOL;
	i 														:	INT;
END_VAR

(* EventHandlingGrp			V4.1	*)
(************************************)

(* status ***************************)
Status  													:= 0;
NoOfActiveEvents											:= 0;

IF(Disable OR SourceId = 0)AND Disabled
THEN
	RETURN;
ELSE
	Disabled												:= Disable OR SourceId = 0;
	
	FOR i := MIN_EVENT TO MAX_EVENT 
	DO
		(* Init Default Class *)
		IF SetClass <> TC2_SYSTEM.TCEVENTCLASS_ALARM
			AND NOT _Mem.7
		THEN
			no[i].eClass										:= SetClass;
			_Mem.7											:= i = MAX_EVENT;
		END_IF                                  			
		                                        			
		IF Disable OR SourceId = 0              			
		THEN                                    			
			no[i].Flag 										:= FALSE;
			no[i].ConfirmTrig 										:= no[i].State <> TCEVENTSTATE_INVALID AND no[i].State <> TCEVENTSTATE_RESETCON;
		ELSIF ConfirmTrig                             			
		THEN                                    	
			no[i].ConfirmTrig 								:= TRUE;
			_Mem.0 											:= ConfirmTrig;
                                                			
		ELSIF _Mem.0                            			
		THEN                                    			
			no[i].ConfirmTrig 								:= FALSE;
			_Mem.0 											:= i <> MAX_EVENT;

		ELSIF AutoConfirm
		THEN
			IF NOT no[i].Flag
				AND no[i].State <> TCEVENTSTATE_INVALID
				AND no[i].State <> TCEVENTSTATE_RESETCON
			THEN
				no[i].ConfirmTrig 							:= TRUE;
			ELSE                                			
				no[i].ConfirmTrig 							:= FALSE;
			END_IF                              			
		END_IF                                  	
                                                	
		(* Mem current Event *)                 	
		IF no[i].State <> TCEVENTSTATE_INVALID OR no[i].Flag 
		THEN
			_Mem.1											:= TRUE;
			(* Call Event *)
			no[i](
				Flag	:= ,
				ConfirmTrig := ,
				MsgId	:= TO_UINT(i + MsgOffset),
				SourceId:= SourceId,
				eClass	:= (* see grp call *),
				Text1	:= (* see grp call *),
				Text2	:= (* see grp call *),
				pText3	:= (* see grp call *),
				State	=> );
		END_IF

		(* Set info flags *)
		IF	no[i].State <> TCEVENTSTATE_INVALID 
		THEN
			NoOfActiveEvents								:= NoOfActiveEvents + 1;
			Status											:= Status OR no[i].Status;
			Disabled										:= FALSE;
		ELSIF _Mem.1
		THEN (* Send one time info event is gone *)
			; 
		END_IF
	END_FOR	
END_IF
(*****************************************************************************************)

METHOD PUBLIC confirm : booL  //Return value = TRUE if execution finished
VAR_INPUT
END_VAR
IF NoOfActiveEvents > 0
THEN
	FOR i := MIN_EVENT TO MAX_EVENT 
	DO
		no[i](ConfirmTrig := TRUE);
	END_FOR
	_Mem.0			:= TRUE;
END_IF

confirm		:= TRUE;
END_METHOD

END_FUNCTION_BLOCK

// POUs/EventLogger/TriggerEvents/EventHandlingStatisticInfo
{attribute 'no_check'}
//Collection with count and class types of active events 
FUNCTION_BLOCK EventHandlingStatisticInfo
VAR_OUTPUT CONSTANT
	MIN_CLASS												: 	UINT := TCEVENTCLASS_NONE;
	MAX_CLASS												: 	UINT := TCEVENTCLASS_PARAMERROR;
	MIN_PRIORITY											: 	INT := 0;
	MAX_PRIORITY											: 	INT := 7;
END_VAR
VAR_INPUT
	ClassInfo												:	ARRAY[MIN_CLASS..MAX_CLASS] OF INT; (* No of active messages in each class
																										TCEVENTCLASS_NONE			:=0
																										TCEVENTCLASS_MAINTENANCE	:=1	
																										TCEVENTCLASS_MESSAGE		:=2
																										TCEVENTCLASS_HINT			:=3	
																										TCEVENTCLASS_STATEINFO		:=4	
																										TCEVENTCLASS_INSTRUCTION	:=5	
																										TCEVENTCLASS_WARNING		:=6	
																										TCEVENTCLASS_ALARM			:=7	
																										TCEVENTCLASS_PARAMERROR		:=8 *)
	PriorityInfo											:	ARRAY[MIN_PRIORITY..MAX_PRIORITY] OF INT; //No of active messages per priority - see Param.EVENT_HANDLING_CONFIG
	NoOfQuitRequiredEvents									:	INT;
	NoOfActiveEvents										:	INT;
END_VAR
VAR_OUTPUT
END_VAR
VAR
	TaskInterlockCountIn									:	BOOL;
	TaskInterlockCountOut									:	BOOL;
END_VAR

;

PROPERTY PUBLIC classAlarmActive : BOOL
GET
classAlarmActive													:= ClassInfo[TCEVENTCLASS_ALARM] <> 0;
END_GET
END_PROPERTY

